// TwinCAT 3 PLC project LCLSVacuum
// Title: LCLSVacuumLib
// Company: SLAC
// Author: Alex Wallace & Scott Stubbs
// ProjectVersion: 1.12.0
// Description: No serial drivers exist in this library. Need LCLSVacuumSerialDrivers for that. 1.2.0 ecat diagnostic 1.2.1 added the ecat lib in here 1.2.2 adding the ratio check function for valve interlocking 1.3.6 added 275 & 500 gauges, minor changes 1.4.0 added a normally open gate valve structure and FB 1.5.0 added error and warning codes to ptm structure for pfeiffers 1.5.1 seamless override open/close on vgc during transition from override to normal mode. 1.7.0 ST_PTM now uses inheritence model. Started implementing Ebara support. 1.8.0 Moved to seperate functions for 937A and 937B controllers.
// ProgramVersion: 3.1.0.9
// libraries:
//   LCLS General,newest,SLAC
//   Tc2_EtherCAT, * (Beckhoff Automation GmbH)
//   Tc2_Standard, * (Beckhoff Automation GmbH)
//   Tc2_System, * (Beckhoff Automation GmbH)
//   Tc2_TcpIp, * (Beckhoff Automation GmbH)
//   Tc2_Utilities, * (Beckhoff Automation GmbH)
//   Tc3_Interfaces, * (Beckhoff Automation GmbH)
//   Tc3_Module, * (Beckhoff Automation GmbH)
// project tree:
//   Data types/Gauges/ E_PressureState.TcDUT, Gauge_Type.TcDUT, ST_VG.TcDUT
//   Data types/IO/ IO_EP2338.TcDUT
//   Data types/ ISG_Struct.TcDUT, ST_Encoder.TcDUT, UpStrInVac_Struct.TcDUT, UpStrOutVac_Struct.TcDUT
//   Data types/Pumps/ E_PumpState.TcDUT, ST_AgilentControlStatus.TcDUT, ST_AgilentPTM.TcDUT, ST_AuxiliaryPump.TcDUT, ST_EbaraDryPump.TcDUT, ST_EbaraPTM.TcDUT, ST_LeyboldPTM.TcDUT, ST_PfeifferPTM.TcDUT, ST_PIP.TcDUT, ST_PTM.TcDUT, ST_ReadbackOnlyPump.TcDUT, ST_RoughPump.TcDUT
//   Data types/Valves/ E_VCN.TcDUT, E_ValvePositionState.TcDUT, E_VGC.TcDUT, ST_VCC.TcDUT, ST_VCC_NO.TcDUT, ST_VCN.TcDUT, ST_VGC.TcDUT, ST_VGC_NO.TcDUT, ST_VRC.TcDUT
//   Global Variables/ Constants.TcGVL, Global_Variables.TcGVL
//   POUs/ Example_GaugeSup.TcPOU
//   POUs/Functions/Gauge FB/ FB_500.TcPOU, FB_903.TcPOU, FB_907.TcPOU, FB_275.TcPOU, FB_909.TcPOU, FB_925.TcPOU, FB_937A_VG.TcPOU, FB_937B_VG.TcPOU, FB_972.TcPOU, FB_Dumb_Gauge.TcPOU, FB_PressureState.TcPOU, FB_GCM.TcPOU, FB_GGO.TcPOU
//   POUs/Functions/Pumps/ FB_EbaraDryPump.TcPOU, FB_PTM_Pfeiffer.TcPOU, FB_PTM_Ebara.TcPOU, FB_PTM_Agilent.TcPOU, FB_PTM_MagDriveDigital.TcPOU, FB_PTM_LeyboldTD20Classic.TcPOU, FB_ScrollPump.TcPOU, FB_TurboExtLogic.TcPOU, FB_VARIAN301TURBO.TcPOU
//   POUs/Functions/Valve FB/ FB_TurbVentvalve_NO.TcPOU, FB_VCC_NO.TcPOU, FB_VCN.TcPOU, FB_VGC.TcPOU, FB_VGC_NO.TcPOU, FB_VRC.TcPOU, FB_VCC.TcPOU, FB_VRC_OK_CLS.TcPOU, F_VALVE_REL_ILK.TcPOU, F_VRC_DIODE_ILK.TcPOU, F_TURBO_VRC_ILK.TcPOU
//   Version/ Global_Version.TcGVL
// real-time tasks:
//   TASK PlcTask: cycle T#10ms, priority 20, ADS port 350
//   TASK LoggerTask: cycle T#10ms, priority 21, ADS port 351

// ---- Data types/Gauges/E_PressureState.TcDUT
TYPE E_PressureState :
(
	//Valid States (Positive)
	Valid := gc_GaugeValidState, // gc_GaugeValidState set in "Global Variable Folder: Constants"
	ValidHi	:= 1, 
	ValidLo	:= 2, 
	
	// Invalid states
	PressInvalid	:= -1, 
	GaugeDisconnected	:=	-2, 
	OoR	:= -6, 
	// Ion gauges
	Off		:= -3, 
	Starting	:= -4
) INT;
END_TYPE

// ---- Data types/Gauges/Gauge_Type.TcDUT
TYPE Gauge_Type: ( 
PG722B := 0, //Baraton Gauge
IG903 := 1 , //Cold Cathode
PG907 := 2 , //Pirani Gauge
IG909:= 3 , //Hot Cathode
PG925 := 4 ); //MicroPirani Gauge
(* This enumeration should match up with the EDM MUX button on the vacuum gauge expert controls screen *)
END_TYPE

// ---- Data types/Gauges/ST_VG.TcDUT
TYPE ST_VG :
STRUCT
	/// A general gauge structure is used to make the rest of the interlocking simpler. There are some parameters for cold cathodes that are not used by pirani.
	///These features aren't disabled, they just aren't used, think child/parent classes. 
	/// Readbacks 
	rPRESS: REAL; //This is the human-readable pressure
	iPRESS_R: INT; //input pressure in machine form
	xAT_VAC: BOOL; //Pressure At Vacuum
	xPRESS_OK: BOOL; // Pressure Reading is trustworthy
	eState	:	E_PressureState;
	
	/// Controls 
	xHV_DIS: BOOL;// Enable High Voltage when True
	xHV_SW: BOOL;// High Voltage Switch
	wHV_RO: WORD;// Relay Output Location
	 // Bakeout bit 
	xBAKEOUT: BOOL;
	//enum for gauge type - will replace iType
	eTYPE: Gauge_Type := Gauge_Type.PG907; 
	//Gauge type, deprecated (default to pirani)
	iTYPE: INT := 2;

	// Index location of the associated Pirani Gauge
	wPG: WORD;  
	
	xTurnOnTime: BOOL;/// Turn on Timers for cold cathode warmup 
	
	rVAC_SP: REAL := 0.5; // At vacuum setpoint for all gauges
	rPRO_SP: REAL := 0.01; // Protection setpoint for ion gauges at which the gauge turns off, not used for pirani
	rHYS_PR: REAL; // Protection setpoint hysteresis 
	rFULL_SCALE: REAL := 1000; // Full scale pressure in Torr for baratron pressure conversion 
END_STRUCT
END_TYPE

// ---- Data types/IO/IO_EP2338.TcDUT
TYPE IO_EP2338 :
STRUCT
	i_bInCh1	AT	%I*	:	BOOL;
	i_bInCh2	AT	%I*	:	BOOL;
	i_bInCh3	AT	%I*	:	BOOL;
	i_bInCh4	AT	%I*	:	BOOL;
	
	i_bInCh5	AT	%I*	:	BOOL;
	i_bInCh6	AT	%I*	:	BOOL;
	i_bInCh7	AT	%I*	:	BOOL;
	i_bInCh8	AT	%I*	:	BOOL;
	
	
	q_bInCh1	AT	%Q*	:	BOOL;
	q_bInCh2	AT	%Q*	:	BOOL;
	q_bInCh3	AT	%Q*	:	BOOL;
	q_bInCh4	AT	%Q*	:	BOOL;

	q_bInCh5	AT	%Q*	:	BOOL;
	q_bInCh6	AT	%Q*	:	BOOL;
	q_bInCh7	AT	%Q*	:	BOOL;
	q_bInCh8	AT	%Q*	:	BOOL;
END_STRUCT
END_TYPE

// ---- Data types/ISG_Struct.TcDUT
TYPE ISG_Struct :
STRUCT

	xdoHV1 : BOOL;
	xdoHV2 : BOOL;
	xdoHV3 : BOOL;

	xswHV1 : BOOL;
	xswHV2 : BOOL;
	xswHV3 : BOOL;

	xilkHV1 : BOOL;
	xilkHV2 : BOOL;
	xilkHV3 : BOOL;

END_STRUCT
END_TYPE

// ---- Data types/Pumps/E_PumpState.TcDUT
TYPE E_PumpState :
(
pumpSTOPPED	:= 0,
pumpSTARTING	:= 1,
pumpRUNNING	:= 2,
pumpFAULT := 3

);
END_TYPE

// ---- Data types/Pumps/ST_AgilentControlStatus.TcDUT
TYPE ST_AgilentControlStatus :
STRUCT

(* Inputs *)
	xdiR1   		:  BOOL;
	xdiLSpd 		:  BOOL;
	xdiStart		:  BOOL;
	xdiR2   		:  BOOL;
	xdiFlt   	:  BOOL;
	xswStart		:  BOOL;
	xswLSpd 		:  BOOL;
	xswSS   		:  BOOL;
	xilkStart	:  BOOL;
	xilkLSpd   	:  BOOL;
	xilkEnb   	:  BOOL;
	xilkSS   	:  BOOL;
	xAlmRst   	:  BOOL;

(* Outputs *)
	xdoStart	:  BOOL;
	xdoLSpd	:  BOOL;
	xdoEnb	:  BOOL;
	xdoSS	:  BOOL;

(* Alarm Outputs *)
	xalmFlt		:  BOOL;
	xalmStart	:  BOOL;
	xalmLSpd		:  BOOL;
	xalmSS		:  BOOL;
	xAlmSum		: BOOL;


END_STRUCT
END_TYPE

// ---- Data types/Pumps/ST_AgilentPTM.TcDUT
TYPE ST_AgilentPTM EXTENDS ST_PTM :
STRUCT

(* Inputs *)
	(* 24V in Ramp state; 0V for others *)
    i_xSTART :	BOOL; 
	
	(* setpoint related to frequency *)
	i_xR1	:  BOOL;
	
	(* setpoint related to Power *)
	i_xR2	:  BOOL;
	
	(* low speed mode *)
	i_xLSpd	:  BOOL;
	
	(* Fault input*)
	//i_xFault : BOOL;  Inherit ST_PTM.xFault
	
	

(* controls *)
	(* Start/Stop - 
		q_RunDo ;   Inherit ST_PTM.
	 *)
	
	(* Low speed control *)
	q_xLSpd		:  BOOL;
	
	(*Soft start *)
	q_xSS   	:  BOOL;
	
	(* Run interlock*)
	q_xIlk : BOOL;
		
	eState	:	E_PumpState;
	
	rForelinePressureSP : REAL := 0.01;
	rInletPressureSP : REAL := 0.5;
	

END_STRUCT
END_TYPE

// ---- Data types/Pumps/ST_AuxiliaryPump.TcDUT
TYPE ST_AuxiliaryPump EXTENDS ST_RoughPump :
STRUCT
	q_ContactClosed	:	BOOL;
END_STRUCT
END_TYPE

// ---- Data types/Pumps/ST_EbaraDryPump.TcDUT
TYPE ST_EbaraDryPump EXTENDS ST_RoughPump :
STRUCT
(* Extension of the rough pump archetype for ebara 
Applicable to: 
EV-S20
EV-S50
EV-S100
EV-S200
*)

//Controls
q_xMPStart	:	BOOL; //Main Pump start
q_xBPStart	:	BOOL; // Booster Pump start (this can be started by the pump automatically)

xBPIlk	:	BOOL;	//Booster pump interlock
rBPIlkSP	:	REAL := 30; //Booster pump pressure setpoint
tonBP	:	TON := (PT:=T#5S); //Timer for pressure and valve stability


//Readbacks
i_xMPStatus	:	BOOL; //MP status
i_xBPStatus	:	BOOL; //BP status
i_xWarning	:	BOOL; //Warning status
i_xAlarm	:	BOOL; //Alarm, maps to error
i_xRemote	:	BOOL; //Remote control status


END_STRUCT
END_TYPE

// ---- Data types/Pumps/ST_EbaraPTM.TcDUT
TYPE ST_EbaraPTM EXTENDS ST_PTM :
STRUCT
(* Extension of the PTM archetype for Ebara turbo controllers 
Applicable to: 
ETC series
*)
//Controls
i_xStart   : BOOL; //Momentary start switch
i_xStop    : BOOL; //Momentary stop switch
// i_xReset is momentary reset switch - resets protection functions

q_xStart   : BOOL; //Outputs - FB decides if these are actually set
q_xStop    : BOOL;
q_xReset   : BOOL;
q_xProtection : BOOL; //NC. If opened, pump will decelerate/not start

iq_xSpeedSet    : BOOL; //Request to set speed
q_iSpeedSet   : DINT; //Requested speed (min. 100 RPM)

i_xOverride   : BOOL; //Override mode - ignores interlocks

//Readbacks - also has Accel/At speed/Decel/Fault/Cur Speed (min 100RPM)
i_xRotate : BOOL; //If open, pump is rotating
i_xDecel  : BOOL; //If closed, brake engaged (pump decelerating)
i_xNCFault  : BOOL; //Normally closed fault wiring. If false, there is a fault, or cable is unplugged.
i_iRawSpeed	:	INT; //Raw pump speed from analog input

END_STRUCT
END_TYPE

// ---- Data types/Pumps/ST_LeyboldPTM.TcDUT
TYPE ST_LeyboldPTM EXTENDS ST_PTM :
STRUCT
(* Extension of the PTM archetype for Oerlikon turbo controllers 
Applicable to: 
Mag Drive Digital
Mag Drive S
More?
*)
//Readbacks
	i_xDecel	:	BOOL;
	i_diPumpTemp:	DINT;
	i_diPwr   	:   DINT;
	i_diElecTemp:	DINT;
	i_xTempFault:	BOOL;
	i_xNCError	:	BOOL; //Using normally closed wiring

//Controls
	q_xRemote : BOOL; (* Remote control enabled *)
END_STRUCT
END_TYPE

// ---- Data types/Pumps/ST_PfeifferPTM.TcDUT
TYPE ST_PfeifferPTM EXTENDS ST_PTM :
STRUCT
(* Extension of the PTM archetype for Pfeiffer turbos 
Applicable to: 
HiPace series w/ onboard controllers
More?
*)
//Readbacks
	i_diPwr		:	DINT;
	i_diElecTemp	:	DINT;
	i_diBtmTemp:	DINT;
	i_diBrngTemp:	DINT;
	i_diMtrTemp:	DINT;
	i_iErrorCode	:	INT; //might change these to enumeration someday
	i_iWarningCode	:	INT;
	i_xTempFault	:	BOOL;
	i_uiPowerPctRbk :   UINT;
	
//Controls
	q_uiPowerPct : UINT := 100; //Should normally be 100
	
END_STRUCT
END_TYPE

// ---- Data types/Pumps/ST_PIP.TcDUT
TYPE ST_PIP :
STRUCT
(* Interlock *)
   xHV_ExtIlk : BOOL; 

	rHVEna_SP : REAL := 1.0E-4;	
	
(* EPICS Controls *)	
	i_xHVEna_SW : BOOL; 
	
(* Controls *)
	q_xHVEna_DO : BOOL;	



END_STRUCT
END_TYPE

// ---- Data types/Pumps/ST_PTM.TcDUT
TYPE ST_PTM :
STRUCT
(* General PTM Structure
Each PTM might have a serial control structure, but all will have a general supervisory control structure

NOTE: This is an archetype, use an extension of this structure for a specific pump (or make one).

*)

(* Controls *)
	i_xRunSW	:	BOOL;
	i_xReset	:	BOOL; //For resetting faults
	q_RunDO 	:	BOOL;

(* Readbacks *)
	xExtRunOk	:	BOOL; (* also a control *)
	i_xAccel	:	BOOL;
	i_xAtSpd	:	BOOL;
	i_diCurSpd	:	DINT;
	
	xCommTimeout	:	BOOL := TRUE;  (* Initialized true since we haven't talked to pump yet *)
(* Alarm Outputs *)
	xFault		:	BOOL; //Note, for Ebara this is *false* in a fault condition!
	xWarn		:	BOOL; (* warning *)
	
(* IWS instructions *)
	xActive	:	BOOL; // this bit is set to add the pump to the system
	iPumpGrp 	:	INT; // all members of a pump group start at the same time
	
(* Operational Setpoints *)
	rForelineSP	:	REAL := 0.5;

END_STRUCT
END_TYPE

// ---- Data types/Pumps/ST_ReadbackOnlyPump.TcDUT
//Simple type for a pump where we have readback only, no control.

TYPE ST_ReadbackOnlyPump :
STRUCT
	i_xPumpOn : BOOL;
	i_diPumpSpeed : DINT; //Arbitrary
END_STRUCT
END_TYPE

// ---- Data types/Pumps/ST_RoughPump.TcDUT
TYPE ST_RoughPump :
STRUCT
	
(* Generic roughing pump controls 

NOTE: This is an archetype, use an extension of this structure for a specific pump (or make one).

*)

//Controls
i_xRunSW	:	BOOL; //epics/ software control switch
q_xRunDo 	:   BOOL; 

//Status and Readback
xIlk	:	BOOL; //Interlock bit, true means OK to run
xExtIlk	:	BOOL; //External interlock, this is where the logic goes
xAtSpd	:	BOOL; //Pump at speed setpoint

xWrn	:	BOOL; //Pump warning
iWrn	:	BOOL; //Warning state/code
xErr	:	BOOL; //Error summary
iErr	:	BOOL; //Error state/code

END_STRUCT
END_TYPE

// ---- Data types/ST_Encoder.TcDUT
TYPE ST_Encoder :
STRUCT
	xENC_PWR_SW : BOOL;
	xENC_PWR : BOOL;
END_STRUCT
END_TYPE

// ---- Data types/UpStrInVac_Struct.TcDUT
TYPE UpStrInVac_Struct :
STRUCT

	xdiUpSVac : BOOL;

END_STRUCT
END_TYPE

// ---- Data types/UpStrOutVac_Struct.TcDUT
TYPE UpStrOutVac_Struct :
STRUCT

	xdoUpSVac : BOOL;
	xilkUpSVac : BOOL;

END_STRUCT
END_TYPE

// ---- Data types/Valves/E_VCN.TcDUT
TYPE E_VCN :
	(
		CloseValve		:= 0,
		OpenValve		:= 2
	);
END_TYPE

// ---- Data types/Valves/E_ValvePositionState.TcDUT
TYPE E_ValvePositionState :
	(
OPEN	:= 0,
CLOSED	:= 1,
MOVING	:= 2,
INVALID :=3
	);
END_TYPE

// ---- Data types/Valves/E_VGC.TcDUT
TYPE E_VGC :
(

	Vented,
	AtVacuum,
	ERR_DiffPress,
	ERR_LostVac

);
END_TYPE

// ---- Data types/Valves/ST_VCC.TcDUT
TYPE ST_VCC :
STRUCT

(* Inputs *)
	xOPN_SW	: BOOL;
	xOvrdOpn	:	BOOL;
	xOPN_OK	: BOOL;

(* Outputs *)
	xOPN_DO	: BOOL;

END_STRUCT
END_TYPE

// ---- Data types/Valves/ST_VCC_NO.TcDUT
TYPE ST_VCC_NO :
STRUCT

(* A normally open valve needs permission to close! *)
(* Inputs *)
	xCLS_SW	: BOOL;
	xOvrdCls	:	BOOL;
	xCLS_OK	: BOOL;

(* Outputs *)
	xCLS_DO	: BOOL;

END_STRUCT
END_TYPE

// ---- Data types/Valves/ST_VCN.TcDUT
TYPE ST_VCN :
STRUCT
	(* VCN - Valve Controlled Needle
	Used for Pfeiffer EVR 116 needle valves *)
	// Inputs
	i_iPosition	:	INT; //Position readback (if it exists)
	
	// Outputs
	q_iRawPosition	:	INT; //Position control 
	//For the EVR 116 this is 0-10V analog
	
	//Softvariables
	xIlk	:	BOOL := FALSE; // Interlock Bit
	rUpperLimit	:	REAL;	//Upper limit on valve open
	rReqPosition	:	REAL; //Requested position (0.0-100.0%)
	eValveControl	:	E_VCN := E_VCN.CloseValve; // Valve control state

	ftIlk	:	F_TRIG;	

END_STRUCT
END_TYPE

// ---- Data types/Valves/ST_VGC.TcDUT
TYPE ST_VGC :
STRUCT

(* Readbacks *)
	i_xOpnLS	: BOOL;
	i_xClsLS	: BOOL;

(* EPICS Controls *)
	xOPN_SW	: BOOL;
	xAlmRst	: BOOL;
	xOvrdOpn	:	BOOL;

(* Interlocks *)
	xDP_OK	:	BOOL;	// Indicates the valve can be opened because the differential pressure is low enough
	xEXT_OK	:	BOOL := FALSE;	(* External interlock for custom interlocking in addition to regular DP ilk, this must be set true, or the interlock condition before calling the FB_VGC *)
	xOPN_OK	:	BOOL;	(* Final SUM of DP_OK and EXT_OK, needed because it allows the DP ilk to be switched off, see FB_VGC.Dis_DPIlk *)
	
	rAT_VAC_SP	:	REAL := 0.01;	// Interlock setpoint for gauges on both sides of valve
	rAT_VAC_SP_LAST	:	REAL :=0.01 ;	// Interlock setpoint for gauges on both sides of valve
	rAT_VAC_HYS	:	REAL :=0.01;	// Hysteresis of the vacuum sp
	rHYST_PERC	:	REAL := 0.80;	// Hysteresis percentage
	xAT_VAC	:	BOOL;	//At vacuum setpoint
	
eState	:	E_ValvePositionState := E_ValvePositionState.INVALID;
(* Controls *)
	xOPN_DO	: BOOL;

(* Alarm Outpus *)
	xERR_DifPres		: 	BOOL;
	xERR_LstVac		: 	BOOL;
	xERR_SM		:	BOOL; //Issue with the valve state-machine. This state should be excluded, if this boolean is true, something dramatic in the PLC software has happened.
	xAlmSum			: 	BOOL;

END_STRUCT
END_TYPE

// ---- Data types/Valves/ST_VGC_NO.TcDUT
TYPE ST_VGC_NO EXTENDS ST_VGC :
STRUCT
	(* A normally open gate valve needs permission to close! *)
	(* EPICS Controls *)
	xCLS_SW	:	BOOL;
	xOvrdCls	:	BOOL;
	
	(* Interlocks *)
	xCLS_OK	:	BOOL;
	
	(* IO Controls *)
	xCLS_DO	:	BOOL;
	
	
END_STRUCT
END_TYPE

// ---- Data types/Valves/ST_VRC.TcDUT
TYPE ST_VRC :
STRUCT
(* Readbacks *)
	//If True, Valve is Open
	i_xOpnLS	:	BOOL;
	//If True, Valve is Closed
	i_xClsLS	:	BOOL;
	
	eState	:	E_ValvePositionState := E_ValvePositionState.INVALID;

(* Inputs *)
	//Manually Pressing valve "Open/Close" on EDM
	xOPN_SW	: BOOL;
	//Manually toggling valve Local "ILK on button" on EDM
	xOvrdOpn	:	BOOL;
	//Calculated permissions to open valve
	xOPN_OK	: BOOL;
	//In case VRC is normally open
	xCLS_OK : BOOL := TRUE;
(* Outputs *)
	//When True, Opens valve
	//When False, Closes valve
	xOPN_DO	: BOOL;

END_STRUCT
END_TYPE

// ---- Global Variables/Constants.TcGVL
VAR_GLOBAL CONSTANT
	gc_iSizeOfGGOArray : INT := 50;
	gc_GaugeValidState :	INT := 0;
END_VAR

// ---- Global Variables/Global_Variables.TcGVL
VAR_GLOBAL
	g_stSystem	:	System_Struct:= (
    	xFirstScan := TRUE
	);
	
	g_DummyVG	:	ST_VG;
	
END_VAR

// ---- Version/Global_Version.TcGVL
{attribute 'TcGenerated'}
// This function has been automatically generated from the project information.
VAR_GLOBAL CONSTANT
	{attribute 'const_non_replaced'}
	{attribute 'linkalways'
	stLibVersion_LCLSVacuumLib : ST_LibVersion := (iMajor := 1, iMinor := 12, iBuild := 0, iRevision := 0, sVersion := '1.12.0');
END_VAR

// ---- POUs/Example_GaugeSup.TcPOU
PROGRAM Example_GaugeSup
VAR

	LMP_VG00	:	ST_VG; (* simulation pirani *)

	fb_LMP_VG :	FB_GGO;
	i : INT;

END_VAR

(* Dummy pirani setup *)
LMP_VG00.rPRESS_OK := TRUE;

(* The following condition ensures that the pressure switches to the GPI:20 when VRC 06 is closed and VRC 05 is open *)

(* Changed interlock here to GPI 20 for running without the GPI 30 gauge *)
(*
IF LMP_VRC05.OPN-DO AND NOT LMP_VRC06.OPN_DO THEN
fb_LMP_GPI_D1(PG := LMP_GPI_D1, PGA := LMP_GPI20, PGB := LMP_GPI01, VICA := LMP_VRC05, VICB := LMP_VRC02);
ELSE
fb_LMP_GPI_D1(PG := LMP_GPI_D1, PGA := LMP_GPI30, PGB := LMP+GPI01, VICA := LMP_VRC06, VICB := LMP_VRC02);
END_IF
*)
(* Dumb Gauge *)
(* fb_LMP_GPI_D1 (PG := LMP_GPI_D1, PGA := LMP_GPI20, PGB := LMP_GPI01, VICA := LMP_VRC05, VICB := LMP_VRC02); *)

LMP_VG[20].VAC_SP := 7.5;
LMP_VG[1].VAC_SP := 1E-1;
LMP_VG[2].VAC_SP := 1E-1;
LMP_VG[12].VAC_SP := 5E-7;

(* Upstream vacuum OK signal *)
(* This signal tells the AMO_PLC that the KBP_VGC_02 is OK to open *)
DiscIO_IC_EB1Ch08 := LMP_VG[12].AT_VAC AND LMP_VGC10.OPN_LS;

(* pnCCD Chamber *)
LMP_VG[40].FULL_SCALE := 1000;
LMP_VG[41].FULL_SCALE := 1;

LMP_VG[1].GAUGE := PG925;
LMP_VG[2].GAUGE := PG925;
LMP_VG[10].GAUGE := PG907;
LMP_VG[11].GAUGE := PG907;
LMP_VG[12].GAUGE := IG903;
LMP_VG[13].GAUGE := IG909;
LMP_VG[20].GAUGE := PG907;
LMP_VG[21].GAUGE := IG903;
LMP_VG[22].GAUGE := IG909;
LMP_VG[30].GAUGE := PG907;
LMP_VG[31].GAUGE := IG903;
LMP_VG[40].GAUGE := PG722B;
LMP_VG[41].GAUGE := IG903;
LMP_VG[42].GAUGE := PG722B;
LMP_VG[43].GAUGE := IG909;

FOR i := 1 TO 50 DO
fb_LMP_VG (index := i, astGauges := LMP_VG);
END_FOR

(*
(* Control function blocks *)

(* Roughing lines *)
fb_LMP_VG01(PG := LMP_VG[1]); (* roughing line *)
fb_LMP_VG02(PG := LMP_VG[2]); (* roots line *)

(* Differential Pumping Chambers *)
(* fb_LMP_GCC10 (IG := LMP_GCC10, PG := LMP_GPI00); *)
(* fb_LMP_GCC11 (IG := LMP_GCC11, PG := LMP_GPI00); *)
fb_LMP_VG10 (PG := LMP_VG[10]);
fb_LMP_VG11 (PG := LMP_VG[11]);

(* Interaction Chamber *)
fb_LMP_VG21 (IG := LMP_VG[21], PG := LMP_VG[20]);
fb_LMP_VG22 (IG := LMP_VG[22], PG := LMP_VG[20]);
fb_LMP_VG20 (PG := LMP_VG[20]);

(* Upstream vacuum OK signal *)
(* This signal tells the AMO_PLC that the KBO_VGC_02 is OK to open *)
DiscIO_IC_EB1Ch08 := LMP_VG[12].AT_VAC AND LMP_VGC10.OPN_LS;

(* Detector Chamber *)
fb_LMP_VG31 (IG := LMP_VG[31], PG := LMP_VG[30]);
fb_LMP_VG30 (PG := LMP_VG[30]);

(* pnCCD Chamber *)
fb_LMP_VG41 (IG := LMP_VG[41], PG := LMP_VG[40]);
fb_LMP_VG43 (IG := LMP_VG[43], PG := LMP_VG[42]);
LMP_VG[40].FULL_SCALE := 1000;
LMP_VG[41].FULL_SCALE := 1;
fb_LMP_VG40 (PG := LMP_VG[40]);
fb_LMP_VG42 (PG := LMP_VG[42]);
*)

END_PROGRAM

// ---- POUs/Functions/Gauge FB/FB_GGO.TcPOU
FUNCTION_BLOCK FB_GGO
VAR_IN_OUT
	iq_astGauges: ARRAY[0..gc_iSizeOfGGOArray] OF ST_VG;
	iq_axHV_RO: ARRAY[0..gc_iSizeOfGGOArray] OF BOOL;
END_VAR
VAR_INPUT
	i_iIndex: INT;
END_VAR
VAR

	stPG: ST_VG;
	stVG: ST_VG;
	//index for associated pirani
	wPG : WORD;

	
	// FBs
	fb903	:	FB_903;
	fb907	:	FB_907;
	fb909	:	FB_909;
	fb925	:	FB_925;
	fbGCM	:	FB_GCM;
	
END_VAR

(* This function block is used to calculate the pressure from the analog input voltage and to provide protection and automatic turn on of ion gauges.
 It also manages the turn on fo the AT_VAC boolean, and checks to make sure the pressure is good *)

(* Full-scale pressure conversion factor *)

(* Real-value voltage calculation *)
(* Generic expression for pressure in the MKS systems

P = 10^(V/0.6-12)

722B = 0
903 = 1
907 = 2
909 = 3
925 = 4

*)

(* Make a copy of gauge at index*)
stVG := iq_astGauges[LIMIT(0 ,i_iIndex, gc_iSizeOfGGOArray)];

(* Check that it is an ion gauge *)
IF stVG.eTYPE = Gauge_Type.IG903 OR stVG.eTYPE = Gauge_Type.IG909 THEN

(* Check that Associated Gauge is within index*)
	IF WORD_TO_INT(stVG.wPG) <= gc_iSizeOfGGOArray THEN
		(* Check pressure gauge type before assignment *)
		(* Add high pressure gauge types here *)
		IF iq_astGauges[stVG.wPG].eTYPE = PG722B OR //722B
		iq_astGauges[stVG.wPG].eTYPE = PG907 OR //907
		iq_astGauges[stVG.wPG].eTYPE = PG925 THEN //925
			stPG := iq_astGauges[stVG.wPG];  (* Copy associated pirani gauge number to local variable *)
		ELSE //Default to allow the IG to turn on, this allows someone to set the PG to another IG and turn the gauge on whenever they want
			stPG.rPRESS := 1E-3;
			stPG.xPRESS_OK := TRUE;
		END_IF
	
	END_IF
END_IF

(* Evaluate each Gauge pressure based on eTYPE*)
CASE iq_astGauges[i_iIndex].eTYPE OF
	
	//Baratron Gauge
	PG722B:
		fbGCM(VG:=iq_astGauges[i_iIndex]);
		
	//Cold Cathode
	Gauge_Type.IG903:
		fb903(IG:=iq_astGauges[i_iIndex], PG:=iq_astGauges[wPG]);
		
	//Pirani Gauge	
	PG907:
		fb907(PG:=iq_astGauges[i_iIndex]);
		
	//Hot Cathode	
	Gauge_Type.IG909:
		fb909(IG:=iq_astGauges[i_iIndex], PG:=iq_astGauges[wPG]);
		
	//MicroPirani Gauge	
	PG925:
		fb925(PG:=iq_astGauges[i_iIndex]);
	ELSE
		(* Now, since we don't know what gauge type we're dealing with, we want 
		to make sure to reset all the gauge parameters, otherwise we may be 
		left with stale information *)
	stVG.rPRESS := 760;
	stVG.xAT_VAC := FALSE;
	stVG.xPRESS_OK := FALSE;
	stVG.xHV_SW := FALSE;
		
END_CASE

(* reAssign "HV On" back into High Voltage Array*)
iq_axHV_RO[LIMIT(0,WORD_TO_INT(stVG.wHV_RO),gc_iSizeOfGGOArray)]:=stVG.xHV_DIS;

END_FUNCTION_BLOCK

// ---- POUs/Functions/Gauge FB/FB_903.TcPOU
FUNCTION_BLOCK FB_903
VAR_IN_OUT

	IG : ST_VG;

END_VAR
VAR_INPUT

	PG : ST_VG;

END_VAR
VAR_OUTPUT
END_VAR
VAR
	rMaxPressure: REAL := 5E-3;
	rMinPressure: REAL := 5E-11; (* Even though spec is 3E-10, manual states that the discharge is off only if output voltage is <0.5V. 
                                    Since this corresponds to ~3.2E-11 torr, let's be safe and call the min. 5E-11. *)

	V: LREAL;
	fbGaugeState : FB_PressureState;
END_VAR

(* This function block is used to provide protection and automatic turn on of ion gauges,
 it also manages the turn on of the AT_VAC boolean, and checks to make sure the pressure is good *)

(* Real-value calculation *)
(* Generic expression for pressure in the MKS systems

P = 10^(V/0.6 -12)

*)

V := 10*INT_TO_LREAL(IG.iPRESS_R)/32767;

IG.rPRESS := LREAL_TO_REAL(EXPT(10,(V-11)));


(* Protection Functions *)
(* If the PG pressure is greater than the IG.PRO_SP then the gauge is disabled *)
(* If the PG pressure is less than the IG.PRO_SP then the gauge is enabled *)
(* This FB also implements some hysteresis so the gauge doesn't have rapid power cycling while near the turn on boundary *)

IF PG.rPRESS <= IG.rPRO_SP AND PG.xPRESS_OK THEN

	IG.xHV_DIS := IG.xHV_SW;

ELSIF IG.xHV_DIS THEN
	IF (IG.rPRESS > (IG.rPRO_SP + IG.rHYS_PR)) OR PG.rPRESS > (IG.rPRO_SP + IG.rHYS_PR) THEN
		IG.xHV_DIS := FALSE;
		IG.xHV_SW := FALSE;
	END_IF
ELSE
	IG.xHV_DIS := FALSE;
	IG.xHV_SW := FALSE;
END_IF

(* Pressure OK check *)
fbGaugeState.i_rV := V;
fbGaugeState.i_MaxPressure := rMaxPressure;
fbGaugeState.i_MinPressure := rMinPressure;
fbGaugeState(iq_stVG:=IG);

//Backwards compatibility
IG.xPRESS_OK := (IG.eState = Valid) OR IG.xBAKEOUT;

(* Setpoint evaluation *)
IG.xAT_VAC := (IG.xPRESS_OK AND (IG.rPRESS<IG.rVAC_SP)) OR IG.xBAKEOUT;

END_FUNCTION_BLOCK

// ---- POUs/Functions/Gauge FB/FB_PressureState.TcPOU
FUNCTION_BLOCK FB_PressureState
VAR_INPUT
	i_rV	:	REAL;
	i_rVMin	:	REAL := 0.01; // Anything less than this voltage is considered disconnected
	i_rVMax :	REAL := 10.5; // Anything more than this is considered invalid
	i_IGTurnOnTime	:	TIME := T#10S;
	
	i_MinPressure	:	REAL;
	i_MaxPressure	:	REAL;
END_VAR
VAR_OUTPUT
	q_eState 	:	E_PressureState;
END_VAR
VAR_IN_OUT
	iq_stVG	:	ST_VG;
END_VAR
VAR
	tonGaugeTurnOnTmr : TON;
END_VAR

(* Pressure State Evaluation
A. Wallace, 2016-8-31

This FB serves to evaluate the state of the pressure based on the raw voltage, pressure, and gauge state.

*)
// Is the gauge plugged in, and within a reasonable range?
IF i_rV < i_rVMin THEN
	q_eState := E_PressureState.GaugeDisconnected;
ELSIF i_rV > i_rVMax THEN
	q_eState := E_PressureState.PressInvalid;
ELSE
	// Is the gauge reading back a pressure that makes sense?
	CASE iq_stVG.eTYPE OF
		Gauge_Type.IG903:
			tonGaugeTurnOnTmr(IN:=iq_stVG.xHV_DIS, PT:=i_IGTurnOnTime, Q=>iq_stVG.xTurnOnTime);
			IF iq_stVG.xHV_DIS THEN
				IF tonGaugeTurnOnTmr.Q THEN
					IF iq_stVG.rPRESS >= i_MinPressure AND iq_stVG.rPRESS <= i_MaxPressure THEN
						q_eState := E_PressureState.Valid;
					ELSE
						q_eState := OoR; 
					END_IF
				ELSE
						q_eState := E_PressureState.Starting;
				END_IF
			ELSE
				q_eState := E_PressureState.Off;
			END_IF
		Gauge_Type.IG909:
			IF iq_stVG.xHV_DIS THEN
				IF iq_stVG.rPRESS >= i_MinPressure AND iq_stVG.rPRESS <= i_MaxPressure THEN
					q_eState := E_PressureState.Valid;
				ELSE
					q_eState := E_PressureState.OoR;
				END_IF
			ELSE
				q_eState := E_PressureState.Off;
			END_IF
		Gauge_Type.PG907, Gauge_Type.PG925, Gauge_Type.PG722B:
			IF iq_stVG.rPRESS >= i_MinPressure AND iq_stVG.rPRESS <= i_MaxPressure THEN
				q_eState := E_PressureState.Valid;
			ELSIF iq_stVG.rPRESS < i_MinPressure THEN
				q_eState := E_PressureState.ValidLo;
			ELSE
				q_eState := E_PressureState.ValidHi;
			END_IF
		ELSE
			q_eState := E_PressureState.PressInvalid;
	END_CASE
END_IF


iq_stVG.eState := q_eState;

// Legacy Press OK boolean eval
iq_stVG.xPRESS_OK := q_eState >= gc_GaugeValidState;

END_FUNCTION_BLOCK

// ---- POUs/Functions/Gauge FB/FB_907.TcPOU
FUNCTION_BLOCK FB_907
VAR_IN_OUT

	PG : ST_VG;

END_VAR
VAR_INPUT
END_VAR
VAR_OUTPUT
END_VAR
VAR
	V : LREAL;
	fbGaugeState : FB_PressureState;
END_VAR
VAR CONSTANT
	A : LREAL := 3.29;
	B : LREAL := 24.98;
	C : LREAL  := 0.98;
	V_0 : LREAL := 0.3752;
	D: LREAL := 4.929;
	F: LREAL := 1.6E-6;
	G: LREAL := -225;
	H: LREAL := 2.0253;
	K: LREAL := 0.52703;
	
	// Torr
	rMaxPressure: REAL := 1000;
	// Torr
	rMinPressure: REAL := 1E-3;
END_VAR

(* This function block is used to provide protection and automatic turn on of ion gauges,
 it also manages the turn on of the AT_VAC boolean, and checks to make sure the pressure is good *)

 //Default setpoint 50 mT
IF PG.rVAC_SP = 0 THEN
	PG.rVAC_SP := 5E-2;
END_IF
 
(* Real-value calculation *)

V := 10*INT_TO_LREAL(PG.iPRESS_R)/32767;

IF V > 0.38 AND V < 4.85 THEN

PG.rPRESS := LREAL_TO_REAL(EXPT((A/(B/(EXPT(V,2)-EXPT(V_0,2)-1))), 1/C));

ELSIF V > 4.85 AND V < 5.18 THEN

PG.rPRESS := LREAL_TO_REAL(SQRT( ( (V-D)+SQRT(EXPT((V-D),2)-4*F*G ))/(2*F) ));

ELSIF V> 5.18 THEN

PG.rPRESS := LREAL_TO_REAL(EXP((V-H)/K));

END_IF

(* Pressure OK check *)
fbGaugeState.i_rV := LREAL_TO_REAL(V);
fbGaugeState.i_MaxPressure := rMaxPressure;
fbGaugeState.i_MinPressure := rMinPressure;
fbGaugeState(iq_stVG:=PG);


(* Setpoint evaluation *)
PG.xAT_VAC := PG.xPRESS_OK AND (PG.rPRESS<PG.rVAC_SP) OR PG.xBAKEOUT;

END_FUNCTION_BLOCK

// ---- POUs/Functions/Gauge FB/FB_909.TcPOU
FUNCTION_BLOCK FB_909
VAR_IN_OUT

	IG : ST_VG;

END_VAR
VAR_INPUT

	PG : ST_VG;

END_VAR
VAR_OUTPUT
END_VAR
VAR
	rMaxPressure: REAL := 5E-2;
	rMinPressure: REAL := 3E-10;

	V: REAL;
	fbGaugeState : FB_PressureState;
END_VAR

(* This function block is used to provide protection and automatic turn on of ion gauges,
 it also manages the turn on of the AT_VAC boolean, and checks to make sure the pressure is good *)

(* Real-value calculation *)
(* Generic expression for pressure in the MKS systems

P = 10^(V/0.6 -12)

*)

V := 10*INT_TO_REAL(IG.iPRESS_R)/32767;

IG.rPRESS := LREAL_TO_REAL(EXPT(10,(V-10)));


(* Protection Functions *)
(* If the PG pressure is greater than the IG.PRO_SP then the gauge is disabled *)
(* If the PG pressure is less than the IG.PRO_SP then the gauge is enabled *)
(* This FB also implements some hysteresis so the gauge doesn't have rapid power cycling while near the turn on boundary *)

IF PG.rPRESS <= IG.rPRO_SP AND PG.xPRESS_OK THEN

	IG.xHV_DIS := IG.xHV_SW;

ELSIF IG.xHV_DIS THEN
	IF IG.rPRESS > IG.rPRO_SP + IG.rHYS_PR OR PG.rPRESS > IG.rPRO_SP + IG.rHYS_PR THEN
		IG.xHV_DIS := FALSE;
		IG.xHV_SW := FALSE;
	END_IF
ELSE
	IG.xHV_DIS := FALSE;
	IG.xHV_SW := FALSE;
END_IF

(* Pressure OK check *)
fbGaugeState.i_rV := V;
fbGaugeState.i_MaxPressure := rMaxPressure;
fbGaugeState.i_MinPressure := rMinPressure;
fbGaugeState(iq_stVG:=IG);

//Backwards compatibility
IG.xPRESS_OK := (IG.eState = Valid) OR IG.xBAKEOUT;

(* Setpoint evaluation *)
IG.xAT_VAC := (IG.xPRESS_OK AND (IG.rPRESS<IG.rVAC_SP)) OR IG.xBAKEOUT;

END_FUNCTION_BLOCK

// ---- POUs/Functions/Gauge FB/FB_925.TcPOU
FUNCTION_BLOCK FB_925
VAR_INPUT
END_VAR
VAR_OUTPUT
END_VAR
VAR_IN_OUT
	PG	: ST_VG;
END_VAR
VAR
	rV : REAL;
	fbGaugeState : FB_PressureState;
	rMaxPressure	:	REAL := 760; //Torr
	rMinPressure	:	REAL := 1E-5; //Torr
END_VAR

(* Standard MKS 9XX series conversion *)
(* works for 972 and 925 *)

//Default setpoint 50 mT
IF PG.rVAC_SP = 0 THEN
	PG.rVAC_SP := 5E-2;
END_IF

rV := 10*INT_TO_REAL(PG.iPRESS_R)/32767;

IF rV >= 0.99 THEN
	IF rV >= 0.99 AND rV < 1 THEN
		PG.rPRESS := 1E-5;
	ELSE
		PG.rPRESS := LREAL_TO_REAL(EXPT(10, REAL_TO_LREAL(rV-6)));
	END_IF
	PG.xPRESS_OK := TRUE; //Backwards compatibility
ELSE
	PG.xPRESS_OK := FALSE;
END_IF

(* Pressure OK check *)
fbGaugeState.i_rV := rV;
fbGaugeState.i_MaxPressure := rMaxPressure;
fbGaugeState.i_MinPressure := rMinPressure;
fbGaugeState(iq_stVG:=PG);

(* Setpoint evaluation *)
PG.xAT_VAC := PG.xPRESS_OK AND (PG.rPRESS < PG.rVAC_SP);

END_FUNCTION_BLOCK

// ---- POUs/Functions/Gauge FB/FB_GCM.TcPOU
FUNCTION_BLOCK FB_GCM
VAR_IN_OUT
	VG	:	ST_VG;
END_VAR
VAR_OUTPUT
END_VAR
VAR
	rMinPressure: REAL;
	rV	:REAL;
END_VAR

(* Baratron Pressure Calc 
A. Wallace
2016-6-16
The full-scale pressure times the ratio of the meas.
voltage to full-scale voltage (10V).
The minimum pressure is always going to be 5e-4 * F.S.V.*)

rMinPressure := VG.rFULL_SCALE * 5E-4;


rV :=MAX((10*INT_TO_REAL(VG.iPRESS_R)/32767),0);
VG.rPRESS := (VG.rFULL_SCALE/10)*rV;
IF VG.rPRESS > rMinPressure THEN
	VG.xPRESS_OK := TRUE;
ELSE
	VG.xPRESS_OK := FALSE;
END_IF

END_FUNCTION_BLOCK

// ---- POUs/Functions/Gauge FB/FB_500.TcPOU
FUNCTION_BLOCK FB_500
VAR_IN_OUT
	IG : ST_VG;
END_VAR
VAR_INPUT
	PG	:	ST_VG;
END_VAR
VAR_OUTPUT
	xHV_SW: BOOL;
	rPRESS: INT;
	rVAC_SP: INT;
END_VAR
VAR
	rV : REAL;
	GaugeTurnOnTmr : TON;
	MinPressure: REAL := 1E-10;
	
END_VAR
VAR CONSTANT
	cDefaultPressure : REAL := 750.0;
	vBase	:	REAL := 0; //corresponding vbase 0V based on default curve.  See manual pg. 44
	pBase	:	REAL := 1.0E-10; //default curve base pressure is 1E-10. Confusing since can't actually read that low using analog out.
	vSlope	:	REAL := 1.0; //looks correct for default curve
END_VAR

(* 500 Logarithmic Output Conversion, factory default configuration *)

rV := 10*INT_TO_REAL(IG.iPRESS_R)/32767;

IF rV >= 0.49 AND rV < 0.6  THEN
	IG.eState := E_PressureState.Starting;
	IG.rPRESS := cDefaultPressure;
ELSIF rV < 0.4 THEN
	IG.eState := E_PressureState.Off;
	IG.rPRESS := cDefaultPressure;
ELSE
	IG.eState := E_PressureState.Valid;
	IG.rPRESS := LREAL_TO_REAL(EXPT(10,((rV-vBase)/vSlope+LOG(pBase))));
END_IF



(* Ion Gauge Protection Functions *)
(* If the PG pressure is greater than the VG.PRO_SP then the gauge is disabled *)
(* If the PG pressure is less than the VG.PRO_SP then the gauge is enabled *)
(* This FB also implements some hysteresis so the gauge doesn't have rapid power cycling while near the turn on boundary *)

IF PG.rPRESS <= IG.rPRO_SP AND PG.xPRESS_OK THEN

	IG.xHV_DIS := IG.xHV_SW;

ELSIF IG.xHV_DIS THEN
	IF IG.rPRESS > (IG.rPRO_SP + IG.rHYS_PR)  OR PG.rPRESS > (IG.rPRO_SP + IG.rHYS_PR) THEN
		IG.xHV_DIS := FALSE;
		IG.xHV_SW := FALSE;
	END_IF
ELSE
	IG.xHV_DIS := FALSE;
	IG.xHV_SW := FALSE;
END_IF

(* Pressure gauge OK checks *)

//Backwards compatibility
IG.xPRESS_OK := (IG.eState = E_PressureState.Valid) OR IG.xBAKEOUT;

(* Setpoint evaluation *)
IG.xAT_VAC := (IG.xPRESS_OK AND (IG.rPRESS < IG.rVAC_SP)) OR IG.xBAKEOUT;

END_FUNCTION_BLOCK

// ---- POUs/Functions/Gauge FB/FB_275.TcPOU
FUNCTION_BLOCK FB_275
VAR_IN_OUT
	PG : ST_VG;
END_VAR
VAR_INPUT
END_VAR
VAR_OUTPUT
END_VAR
VAR

	MinPressure: REAL := 1E-4;

	V : REAL;

	Vlowest: REAL := 10;
END_VAR
VAR CONSTANT
	rValidLoBoundary	:	REAL := 0.38;
	rDisconnectedBoundary	:	REAL := 0.3;
END_VAR

(* This function block is used to provide protection and automatic turn on of ion gauges,
 it also manages the turn on of the AT_VAC boolean, and checks to make sure the pressure is good *)
(* For MKS 275 mini-convectron *)

 //Default setpoint 50 mT
IF PG.rVAC_SP = 0 THEN
	PG.rVAC_SP := 5E-2;
END_IF

(* Real-value calculation *)

V := 10*INT_TO_REAL(PG.iPRESS_R)/32767;	

Vlowest := MIN(V, Vlowest);

IF V > rDisconnectedBoundary AND V <= rValidLoBoundary THEN

PG.rPRESS := MinPressure;
PG.eState := ValidLo;

ELSIF V > rValidLoBoundary AND V < 2.842 THEN

PG.rPRESS := MAX( MinPressure, LREAL_TO_REAL( -0.02585 + 0.03767*V + 0.04563*EXPT(V,2)+ 0.1151*EXPT(V,3) - 0.04158*EXPT(V,4)+ 0.008737*EXPT(V,5)) );
PG.eState := Valid;

ELSIF V >= 2.842 AND V < 4.945 THEN

PG.rPRESS := LREAL_TO_REAL((0.1031-0.02322*V+0.07229*EXPT(V,2))/(1-0.3986*V+0.07438*EXPT(V,2)-0.006866*EXPT(V,3)));
PG.eState := Valid;

ELSIF V >= 4.945 AND V < 5.659 THEN

PG.rPRESS := LREAL_TO_REAL((100.624-20.5623*V)/(1-0.37679*V+0.0348656*EXPT(V,2)));
PG.eState := Valid;

ELSIF V <= rDisconnectedBoundary THEN

PG.eState := E_PressureState.GaugeDisconnected; //Most likely not connected
PG.rPRESS := -1;

ELSE
	
PG.eState := OoR; //Larger voltage, probably out of range?
PG.rPRESS := -1;

END_IF


(* Pressure OK check *)
PG.xPRESS_OK := (PG.rPRESS >= MinPressure) AND (PG.eState >= 0);//Make sure to evaluate eState Too!!!!

(* Setpoint evaluation *)
PG.xAT_VAC := PG.xPRESS_OK AND (PG.rPRESS<PG.rVAC_SP);

END_FUNCTION_BLOCK

// ---- POUs/Functions/Gauge FB/FB_937A_VG.TcPOU
FUNCTION_BLOCK FB_937A_VG
VAR_IN_OUT
	VG : ST_VG;
END_VAR
VAR_INPUT
	PG	:	ST_VG := g_DummyVG;
END_VAR
VAR_OUTPUT
END_VAR
VAR
	rV	:	LREAL;
END_VAR

(* 937A Logarithmic Output Conversion *)
(* 7-15-2015 *)
(* This function will read the pressure from any gauge on a 937A. *)

rV := LREAL#10*INT_TO_LREAL(VG.iPRESS_R)/LREAL#32767;
VG.rPRESS := LREAL_TO_REAL(EXPT(10,rV/LREAL#0.6-LREAL#12));


(* Ion Gauge Protection Functions *)
(* If the PG pressure is greater than the VG.PRO_SP then the gauge is disabled *)
(* If the PG pressure is less than the VG.PRO_SP then the gauge is enabled *)
(* This FB also implements some hysteresis so the gauge doesn't have rapid power cycling while near the turn on boundary *)

IF PG.rPRESS < VG.rPRO_SP THEN

VG.xHV_DIS := NOT VG.xHV_SW;

ELSIF NOT VG.xHV_DIS THEN
	IF VG.rPRESS > VG.rPRO_SP + VG.rHYS_PR OR PG.rPRESS > VG.rPRO_SP + VG.rHYS_PR THEN
		VG.xHV_DIS := TRUE;
	END_IF
ELSE
	VG.xHV_DIS := TRUE;
END_IF


(* Pressure gauge OK checks *)
VG.xPRESS_OK := (rV <=9.6 ) AND (rV>=0.6); //legacy

IF (rV <=9.6 ) AND (rV>=0.6) THEN
	VG.eState := E_PressureState.Valid; // normal
ELSIF rV >= 0.18 AND rV <= 0.22 THEN
	VG.eState := E_PressureState.ValidLo; //LO
ELSIF rV >= 9.7 AND rV<= 9.9 THEN
	VG.eState := E_PressureState.ValidHi; //HIGH
ELSIF rV < 0.18 THEN
	VG.eState := E_PressureState.GaugeDisconnected; //not on
ELSE
	VG.eState := E_PressureState.PressInvalid; //other fault - could be no gauge, controller powering up etc
END_IF

(* Setpoint evaluation *)
VG.xAT_VAC := (VG.eState = E_PressureState.Valid) AND VG.rPRESS < VG.rVAC_SP;

END_FUNCTION_BLOCK

// ---- POUs/Functions/Gauge FB/FB_937B_VG.TcPOU
FUNCTION_BLOCK FB_937B_VG
VAR_IN_OUT
	VG : ST_VG;
END_VAR
VAR_INPUT
	PG	:	ST_VG := g_DummyVG;
END_VAR
VAR_OUTPUT
END_VAR
VAR
	rV	:	REAL;
END_VAR

(* 937B Logarithmic Output Conversion *)
(* 5-20-2016, Alex Wallace and Scott Stubbs *)
(* This function will read the pressure from any gauge on a 937B. *)

rV := 10*INT_TO_REAL(VG.iPRESS_R)/32767;
VG.rPRESS := LREAL_TO_REAL(EXPT(10,(rV-7.2)/0.6));


(* Ion Gauge Protection Functions *)
(* If the PG pressure is greater than the VG.PRO_SP then the gauge is disabled *)
(* If the PG pressure is less than the VG.PRO_SP then the gauge is enabled *)
(* This FB also implements some hysteresis so the gauge doesn't have rapid power cycling while near the turn on boundary *)

IF PG.rPRESS < VG.rPRO_SP THEN

VG.xHV_DIS := NOT VG.xHV_SW;

ELSIF NOT VG.xHV_DIS THEN
	IF VG.rPRESS > VG.rPRO_SP + VG.rHYS_PR OR PG.rPRESS > VG.rPRO_SP + VG.rHYS_PR THEN
		VG.xHV_DIS := TRUE;
	END_IF
ELSE
	VG.xHV_DIS := TRUE;
END_IF


(* Pressure gauge OK checks *)
VG.xPRESS_OK := (rV <=9.6 ) AND (rV>=0.6);

IF (rV <=9.7 ) AND (rV>=0.3) THEN
	VG.eState := Valid; // normal
ELSIF rV >= 0.18 AND rV <= 0.22 THEN
	VG.eState := ValidLo; //LO
ELSIF rV > 9.7 AND rV<= 9.9 THEN
	VG.eState := ValidHi; //HIGH
ELSIF rV < 0.18 THEN
	VG.eState := E_PressureState.GaugeDisconnected; //not on
ELSE
	VG.eState := PressInvalid; //other fault - could be no gauge, controller powering up etc
END_IF

(* Setpoint evaluation *)
VG.xAT_VAC := (VG.eState =Valid) AND VG.rPRESS < VG.rVAC_SP;

END_FUNCTION_BLOCK

// ---- POUs/Functions/Gauge FB/FB_972.TcPOU
FUNCTION_BLOCK FB_972
VAR_INPUT
END_VAR
VAR_OUTPUT
END_VAR
VAR_IN_OUT
	VG	: ST_VG;
END_VAR
VAR
	rV : LREAL;
END_VAR

(* Standard MKS 9XX series conversion *)
(* works for 972 and 925 *)

rV := 10*INT_TO_LREAL(VG.iPRESS_R)/32767;

IF rV > 1 THEN
	VG.rPRESS := LREAL_TO_REAL(EXPT(10, 2*rV-11));
	VG.xPRESS_OK := TRUE;
	VG.eState := Valid; //Press OK
ELSE
	VG.xPRESS_OK := FALSE;
	VG.eState := -6;
END_IF

END_FUNCTION_BLOCK

// ---- POUs/Functions/Gauge FB/FB_Dumb_Gauge.TcPOU
FUNCTION_BLOCK FB_Dumb_Gauge
VAR_IN_OUT
	iq_stPG : ST_VG;
END_VAR
VAR_INPUT
	i_stPGA : ST_VG;
	i_stPGB : ST_VG;
	i_stVRCA : ST_VRC;
	i_stVRCB : ST_VRC;
END_VAR
VAR_OUTPUT
END_VAR
VAR
END_VAR

(*
Alex Wallace 2013-10-28

The dummy gauge functions like so:
If my A side valve is open, I mimic the A side gauge.
If my B 	"	 			"			B	"		.
Else, I am at atmosphere, and my pressure is OK. 

The point of this gauge is to provide pressure readbacks for sections of the line that do not have gauges, and may move into an unknown pressure state.
*)

IF i_stVRCA.xOPN_DO THEN
iq_stPG := i_stPGA;
ELSIF i_stVRCB.xOPN_DO THEN
iq_stPG := i_stPGB;
ELSE
iq_stPG.xAT_VAC := FALSE;
iq_stPG.rPRESS := 750;
iq_stPG.xPRESS_OK := TRUE;
END_IF

END_FUNCTION_BLOCK

// ---- POUs/Functions/Pumps/FB_EbaraDryPump.TcPOU
FUNCTION_BLOCK FB_EbaraDryPump
VAR_INPUT
	i_stBPGauge	:	ST_VG; //booster pump interlock gauge
	i_xVlvOpn	:	BOOL; //valve(s) to main system load are open
END_VAR
VAR_OUTPUT
END_VAR
VAR_IN_OUT
	stPump	:	ST_EbaraDryPump; //Ebara dry pump structure
END_VAR
VAR
END_VAR

(* Ebara Dry Pump Control Routine
A. Wallace
2016-4-29
Applicable to:
EV-S20
EV-S50
EV-S100
EV-S200

Does basic controls for the pump. Starts booster pump when appropriate. Turns off pump
in the event of errors/ warnings. Provides interlocking interface.

Main Pump Operational Note:
Ebara recommends that the pump be exposed to the full system load after the main pump is running.

Booster Pump Operational Note:
The booster pump can either be started automatically by the pump itself (probably based on a timer?)
or it can be started by the PLC. The pressure setpoint is by default 30T. It may be wise to make
sure the pump was exposed to the full system load before starting the booster.

*)

//Mapping

// These are normally closed inputs
stPump.xErr := NOT stPump.i_xAlarm;
stPump.xWrn := NOT stPump.i_xWarning;


//Interlock and error/warning
stPump.xIlk :=  stPump.xExtIlk AND NOT (stPump.xErr OR stPump.xWrn);

//Start/ Stop the pump
IF stPump.xIlk THEN
	stPump.q_xMPStart := stPump.i_xRunSW;
ELSE
	stPump.q_xMPStart := stPump.i_xRunSW := FALSE;
END_IF

//Booster pump
stPump.xBPIlk := i_xVlvOpn AND stPump.i_xMPStatus AND (i_stBPGauge.rPRESS < stPump.rBPIlkSP) AND i_stBPGauge.xPRESS_OK;
stPump.tonBP(IN:=stPump.xBPIlk);
stPump.q_xBPStart := stPump.tonBP.Q;

END_FUNCTION_BLOCK

// ---- POUs/Functions/Pumps/FB_PTM_Pfeiffer.TcPOU
FUNCTION_BLOCK FB_PTM_Pfeiffer
VAR_IN_OUT
	iq_stPTM : ST_PfeifferPTM;
END_VAR
VAR_INPUT
END_VAR
VAR_OUTPUT
END_VAR
VAR
END_VAR

(* Basic pump supervisory section *)
IF iq_stPTM.xExtRunOk AND NOT (iq_stPTM.xFault OR iq_stPTM.i_xTempFault) THEN
	iq_stPTM.q_RunDO:=iq_stPTM.i_xRunSW;
ELSE
	iq_stPTM.i_xRunSW:=0;
	iq_stPTM.q_RunDO:=FALSE;
END_IF

END_FUNCTION_BLOCK

// ---- POUs/Functions/Pumps/FB_PTM_Ebara.TcPOU
FUNCTION_BLOCK FB_PTM_Ebara
VAR_IN_OUT
	iq_stPTM : ST_EbaraPTM;
END_VAR
VAR_INPUT
	i_iADCBits : UINT := 15;
	i_iRawSpeed: INT; //Should come from PLC Soft IO.
END_VAR
VAR_OUTPUT
END_VAR
VAR
	TOF_START: TOF := (PT:=T#0.5S); //Manual states momentary switches need to be closed for >= 0.3s
	TOF_STOP: TOF := (PT:=T#0.5S);
	TOF_RESET: TOF :=(PT:=T#0.5S);
END_VAR

(* Ebara ETC control FB
Scott Stubbs & Alex W.
*)

(* Switch processing *)
TOF_START.IN := iq_stPTM.i_xStart;
TOF_START();
TOF_STOP.IN  := iq_stPTM.i_xStop;
TOF_STOP();
TOF_RESET.IN := iq_stPTM.i_xReset;
TOF_RESET();

//Normally closed fault handling
iq_stPTM.xFault := NOT iq_stPTM.i_xNCFault;

(* Simple protection reset *)
IF iq_stPTM.xExtRunOk THEN
	iq_stPTM.q_xProtection:=TRUE;
END_IF

(* Basic pump supervisory section *)
	(* If override mode, ignore everything else *)
IF iq_stPTM.i_xOverride THEN
	IF TOF_START.Q THEN
	iq_stPTM.q_RunDO:=TRUE;
	ELSIF TOF_STOP.Q THEN
		iq_stPTM.q_RunDO:=FALSE;
	END_IF
	//Handle faults - the way the Ebara cable is done, xFault is normally closed
ELSIF iq_stPTM.xFault OR (iq_stPTM.q_RunDO AND NOT iq_stPTM.xExtRunOk) THEN
	iq_stPTM.q_RunDO:=FALSE;
	iq_stPTM.q_xProtection:=FALSE;
	//And one for when we need to start the pump normally. Only allows pump to be started if ILK ok.
ELSIF TOF_START.Q AND iq_stPTM.xExtRunOk THEN
	iq_stPTM.q_RunDO:=TRUE;
	iq_stPTM.q_xStart:=TOF_START.Q;
//One section for when pump is told to stop
ELSIF TOF_STOP.Q THEN
		iq_stPTM.q_RunDO:=FALSE;
END_IF 

iq_stPTM.q_xReset:=TOF_RESET.Q; //No need for a conditional on these, code below takes care of it
iq_stPTM.q_xStop:=TOF_STOP.Q;
//Reset the start switch after processing
IF iq_stPTM.q_RunDO THEN
	iq_stPTM.q_xStart := TOF_START.Q;
END_IF

(* Pump speed calculation *)
IF iq_stPTM.i_iRawSpeed / (EXPT(2,i_iADCBits)-1) * 10 >= 0.2 THEN //Speed reading appears to zero at ~0.16V
iq_stPTM.i_diCurSpd := LREAL_TO_DINT(iq_stPTM.i_iRawSpeed/(EXPT(2,i_iADCBits)-1)*67000);
//V (AI/(2^{# ADC bits} -1 ) * 10[ADC 10V scaling]) * (33600 [Max RPM] - 100) / 5
ELSE
	iq_stPTM.i_diCurSpd := 0;
END_IF

END_FUNCTION_BLOCK

// ---- POUs/Functions/Pumps/FB_PTM_Agilent.TcPOU
FUNCTION_BLOCK FB_PTM_Agilent
VAR_IN_OUT
	iq_stPTM	:	ST_AgilentPTM;
END_VAR
VAR_INPUT
END_VAR
VAR_OUTPUT
END_VAR
VAR
	
END_VAR

(* Basic Agilent Turbo Controls *)
(* A. Wallace, 2015-7-15 *)

(* Pump state *)
(* If frequency (R1) is not above setpoint and pump is not Starting, pump estate is STOPPED, 
   else if frequency (R1) is not above setpoint and pump is Starting, pump estate is STARTING, 
	else if frequency (R1) is above setpoint and pump is not Starting, pump estate is STOPPED, 
*)
IF iq_stPTM.xFault THEN 
	iq_stPTM.eState := E_PumpState.pumpFAULT;

ELSIF NOT iq_stPTM.i_xR1 AND NOT iq_stPTM.i_xSTART  THEN
	iq_stPTM.eState := E_PumpState.pumpSTOPPED;
ELSIF NOT iq_stPTM.i_xR1 AND iq_stPTM.i_xSTART  THEN
	iq_stPTM.eState := E_PumpState.pumpSTARTING;
ELSIF iq_stPTM.i_xR1 AND NOT iq_stPTM.i_xSTART THEN
	iq_stPTM.eState := E_PumpState.pumpRUNNING;
ELSE 
	iq_stPTM.eState := E_PumpState.pumpFAULT;
END_IF

(* Interlock Sum *)
iq_stPTM.q_xIlk := iq_stPTM.xExtRunOk AND NOT iq_stPTM.xFault;

(* Basic pump supervisory section *)
IF iq_stPTM.q_xIlk THEN
	iq_stPTM.q_RunDO := iq_stPTM.i_xRunSW;
ELSE
	iq_stPTM.i_xRunSW:=FALSE;
	iq_stPTM.q_RunDO:=FALSE;
END_IF

(* Mask the at speed bit if fault is true 
done for versions of the interface cable where
at speed gets its power from from the beckhoff term*)

(*Basically if Fault, then squash everything and turn everything off*)
IF iq_stPTM.xFault THEN
	iq_stPTM.i_xAtSpd := FALSE;
	iq_stPTM.i_xRunSW:=FALSE;
	iq_stPTM.q_RunDO:=FALSE;
	iq_stPTM.q_xSS := FALSE;
	iq_stPTM.q_xLSpd:= FALSE;
	iq_stPTM.eState := E_PumpState.pumpFAULT;
END_IF

END_FUNCTION_BLOCK

// ---- POUs/Functions/Pumps/FB_PTM_MagDriveDigital.TcPOU
FUNCTION_BLOCK FB_PTM_MagDriveDigital
VAR_IN_OUT
	iq_stPTM	:	ST_LeyboldPTM;
END_VAR
VAR_INPUT
END_VAR
VAR_OUTPUT
END_VAR
VAR
	xRunOk	:	BOOL;
	tofRemoteDelay	:	TOF;
	
END_VAR

(* Basic MagDrive Digital Turbo Controls *)
(* A. Wallace, 2015-7-15 *)

tofRemoteDelay(IN:=iq_stPTM.q_RunDO, PT:=T#5S);

iq_stPTM.q_xRemote := tofRemoteDelay.Q;

(* Interlock Sum *)
xRunOk := iq_stPTM.xExtRunOk AND NOT iq_stPTM.xFault;

(* Basic pump supervisory section *)
IF xRunOk THEN
	iq_stPTM.q_RunDO := iq_stPTM.i_xRunSW;
ELSE
	iq_stPTM.i_xRunSW:=FALSE;
	iq_stPTM.q_RunDO:=FALSE;
END_IF

END_FUNCTION_BLOCK

// ---- POUs/Functions/Pumps/FB_PTM_LeyboldTD20Classic.TcPOU
FUNCTION_BLOCK FB_PTM_LeyboldTD20Classic
VAR_IN_OUT
	iq_stPTM : ST_LeyboldPTM;
END_VAR
VAR_INPUT
END_VAR
VAR_OUTPUT
END_VAR
VAR
	rtReset	:	R_TRIG;
END_VAR

(* Leybold TD20 Classic FB
A. Wallace
NOTE: This FB should be instanced for each pump. It relies on a
persistent state for reseting faults.
*)

//Faults
	rtReset(CLK:=iq_stPTM.i_xReset);
	iq_stPTM.xFault R= rtReset.Q;
	iq_stPTM.xFault S= iq_stPTM.i_xTempFault OR NOT iq_stPTM.i_xNCError;

	iq_stPTM.xWarn R= rtReset.Q;
	iq_stPTM.xWarn S= iq_stPTM.xCommTimeout;

(* Basic pump supervisory section *)
IF iq_stPTM.xExtRunOk AND NOT iq_stPTM.xFault THEN
	iq_stPTM.q_RunDO:=iq_stPTM.i_xRunSW;
ELSE
	iq_stPTM.i_xRunSW:=FALSE;
	iq_stPTM.q_RunDO:=FALSE;
END_IF

END_FUNCTION_BLOCK

// ---- POUs/Functions/Pumps/FB_ScrollPump.TcPOU
FUNCTION_BLOCK FB_ScrollPump
VAR_IN_OUT
	iq_stPFO	:	ST_RoughPump;
END_VAR
VAR_INPUT
	TurboIsON : BOOL;
	VentValve	: ST_VCC_NO;
END_VAR
VAR
	Tmr_TOF : TOF;
END_VAR

//Turn on scroll pump if the Turbo Vent Valve is closed. So you are not just
// pumping air and accomplishing nothing

// cannot turn off scroll pump if turb is running. delay scroll off 150s.  


Tmr_TOF(IN:=TurboIsON, PT := T#150S);

IF VentValve.xCLS_DO THEN
	iq_stPFO.q_xRunDo := (Tmr_TOF.Q OR iq_stPFO.i_xRunSW);
ELSE
	iq_stPFO.q_xRunDo := FALSE;
END_IF

iq_stPFO.i_xRunSW := iq_stPFO.q_xRunDo;

END_FUNCTION_BLOCK

// ---- POUs/Functions/Pumps/FB_TurboExtLogic.TcPOU
FUNCTION_BLOCK FB_TurboExtLogic
VAR_IN_OUT
	Turbo		:	ST_AgilentPTM;
END_VAR
VAR_INPUT
	BackingGauge:	ST_VG;
	InletGauge	:	ST_VG;
	VentValve	:	ST_VCC_NO;
	ScrollPump	:	ST_RoughPump;
END_VAR
VAR_OUTPUT
END_VAR
VAR
END_VAR

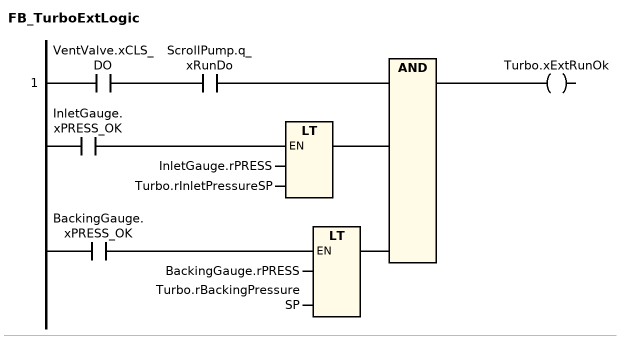
// NETWORK 1
Turbo.xExtRunOk := (VentValve.xCLS_DO AND ScrollPump.q_xRunDo) AND (InletGauge.xPRESS_OK AND InletGauge.rPRESS < Turbo.rInletPressureSP) AND (BackingGauge.xPRESS_OK AND BackingGauge.rPRESS < Turbo.rBackingPressureSP);

END_FUNCTION_BLOCK

// ---- POUs/Functions/Pumps/FB_VARIAN301TURBO.TcPOU
FUNCTION_BLOCK FB_VARIAN301TURBO

VAR_INPUT

	i_xglbAlmRst : BOOL;

END_VAR

VAR

	StartAlmTmr 	: TON;
	LSpdAlmTmr  	: TON;
	SSAlmTmr		: TON;
	tAlmDly			: TIME;

	xStartAlmFlag 	: BOOL;
	xLSpdAlmFlag  	: BOOL;
	xSSAlmFlag		: BOOL;

	xEND: BOOL;
END_VAR

VAR_IN_OUT

	iq_stTP: ST_PTM;

END_VAR

(* Resolve Interlocks *)
(* If Start Ilk is satisfied, other Ilk's are satisfied as well. *)

	iq_stTP.ilkEnb 	:= iq_stTP.ilkStart;
	iq_stTP.ilkLSpd	:= iq_stTP.ilkStart;
	iq_stTP.ilkSS	:= iq_stTP.ilkStart;

(* Hardware Enable Logic & Switch Feedback  *)
	IF NOT iq_stTP.ilkStart THEN
		iq_stTP.swStart := FALSE;
		iq_stTP.swLSpd := FALSE;
		iq_stTP.swSS := FALSE;
		iq_stTP.doEnb := FALSE;
	ELSE
		iq_stTP.doEnb := TRUE;
	END_IF;

(* Pump Control *)
	IF iq_stTP.doEnb THEN
		iq_stTP.doStart := iq_stTP.swStart;
		iq_stTP.doLSpd := iq_stTP.swLSpd;
		iq_stTP.doSS := iq_stTP.swSS;
	ELSE
		iq_stTP.doStart := FALSE;
		iq_stTP.doLSpd := FALSE;
		iq_stTP.doSS := FALSE;
	END_IF

(* ALARM SECTION *)
(* Standard Delay 30 minutes *)
tAlmDly := T#4m;

(* Fail To Start Alarm *)
xStartAlmFlag := iq_stTP.doStart AND NOT iq_stTP.diR1;
IF iq_stTP.doStart AND NOT iq_stTP.almStart THEN
	StartAlmTmr(IN:=xStartAlmFlag, PT:=tAlmDly, Q=>iq_stTP.almStart);
END_IF;
iq_stTP.AlmStart := iq_stTP.almStart AND NOT (i_xglbAlmRst OR iq_stTP.AlmRst);

(* Low Speed Failure Alarm *)
xLSpdAlmFlag := iq_stTP.doLSpd AND NOT iq_stTP.diLSpd;
IF iq_stTP.doLSpd AND NOT iq_stTP.almLSpd THEN
	LSpdAlmTmr(IN:=xLSpdAlmFlag, PT:=tAlmDly, Q=>iq_stTP.almLSpd);
END_IF;
iq_stTP.AlmLSpd := iq_stTP.AlmLSpd AND NOT (i_xglbAlmRst OR iq_stTP.AlmRst);

(* Soft Start Failure Alarm *)
xSSAlmFlag := iq_stTP.doSS AND NOT iq_stTP.diR1;
IF iq_stTP.doSS AND NOT iq_stTP.almSS THEN
	SSAlmTmr(IN:=xSSAlmFlag, PT:=tAlmDly, Q=>iq_stTP.almSS);
END_IF;
iq_stTP.AlmSS := iq_stTP.AlmSS AND NOT (i_xglbAlmRst OR iq_stTP.AlmRst);

(* Alarm Summary - Set the Alarm Summary flag if any alarm is active. *)
iq_stTP.AlmSum := iq_stTP.almFlt OR iq_stTP.almLSpd OR iq_stTP.AlmRst OR iq_stTP.almSS OR iq_stTP.almStart;

END_FUNCTION_BLOCK

// ---- POUs/Functions/Valve FB/FB_TurbVentvalve_NO.TcPOU
FUNCTION_BLOCK FB_TurbVentvalve_NO
VAR_IN_OUT
	iq_stValve : ST_VCC_NO;
END_VAR
VAR_INPUT
	i_stPTM	: ST_AgilentPTM;
END_VAR
VAR
	tofTmr 		: 	TOF;
END_VAR

(*If the turbo is on, you cannot open the valve. In order to open the valve, you have to allow the turbopump
 to have already been turned off for 2 minutes and you have to press the open button on the vent valve

If the code looks confusing please use a truth table to verify*)

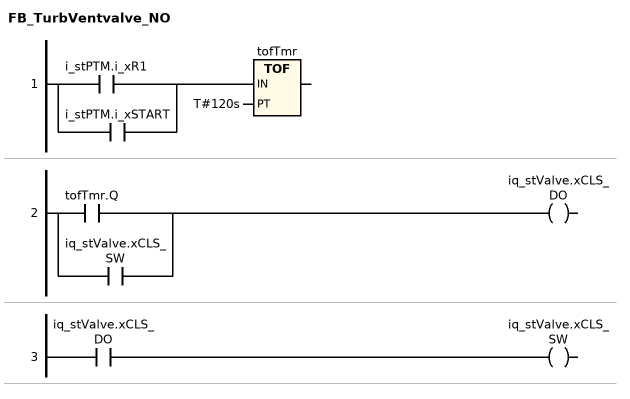
// NETWORK 1
tofTmr(IN := i_stPTM.i_xR1 OR i_stPTM.i_xSTART, PT := T#120s); // TOF

// NETWORK 2
iq_stValve.xCLS_DO := tofTmr.Q OR iq_stValve.xCLS_SW;

// NETWORK 3
iq_stValve.xCLS_SW := iq_stValve.xCLS_DO;

END_FUNCTION_BLOCK

// ---- POUs/Functions/Valve FB/FB_VCC_NO.TcPOU
FUNCTION_BLOCK FB_VCC_NO
VAR_IN_OUT

	iq_stValve : ST_VCC_NO;

END_VAR
VAR_INPUT

END_VAR
VAR_OUTPUT
END_VAR
VAR

tonOvrd	:	TON;
tonDelOK : TON;
rtOK	:	R_TRIG;

END_VAR


IF NOT iq_stValve.xCLS_OK THEN
iq_stValve.xCLS_SW := FALSE;
END_IF

(* Override logic *)
(* Goal: give ability to override, but do so in a way that people won't forget it.
Solution: Override only after ten seconds of override, protect against blips,
when the valve permission goes true for more than ten seconds consistently, remove override
*)

tonDelOK(IN:=iq_stValve.xCLS_OK, PT:=T#10S);
rtOK(CLK:=tonDelOK.Q);
IF rtOK.Q THEN iq_stValve.xOvrdCls :=FALSE; END_IF

//Override timer
tonOvrd(IN:=iq_stValve.xOvrdCls, PT:=T#10S);

(* Here's where the valve is closed *)
iq_stValve.xCLS_DO := (iq_stValve.xCLS_SW AND iq_stValve.xCLS_OK) OR (tonOvrd.Q AND g_stSystem.xOverrideMode);

END_FUNCTION_BLOCK

// ---- POUs/Functions/Valve FB/FB_VCN.TcPOU
FUNCTION_BLOCK FB_VCN
VAR_INPUT
	i_xExtIlk	:	BOOL; //External Interlock
	i_ReqPos	:	BOOL; //Requested position
END_VAR
VAR_OUTPUT
END_VAR
VAR_IN_OUT
	iq_stVCN	:	ST_VCN; //Needle valve structure
END_VAR
VAR
	// Requested voltage
	rReqVoltage: REAL := 0;
END_VAR
VAR CONSTANT
	rOpenVoltage	:	REAL := 9.1; // From the EVR 116 manual
	rCloseVoltage	:	REAL := 0.4;
END_VAR

(* Needle valve control FB
A. Wallace 2016-7-21

This FB should be used as a low level control block.

It provides:

Valve position ceiling
Interlock
Scaling

It is not intended for:
Closed-loop control

It could be used for:
Valve position/flow linearization

Note: Raw position calc is based on 0.5 to 9V span, 32767 bits
*)




// Interlocking
iq_stVCN.xIlk := i_xExtIlk;

IF iq_stVCN.xIlk THEN
	
	IF iq_stVCN.eValveControl = OpenValve THEN
		iq_stVCN.rReqPosition := iq_stVCN.rUpperLimit;
	ELSIF iq_stVCN.eValveControl = E_VCN.CloseValve THEN
		iq_stVCN.rReqPosition := 0;
	END_IF

	//Raw position calc
	iq_stVCN.rReqPosition := LIMIT(0, iq_stVCN.rReqPosition, iq_stVCN.rUpperLimit);
	rReqVoltage := iq_stVCN.rReqPosition * (rOpenVoltage-rCloseVoltage)/100 + rCloseVoltage;
	rReqVoltage := LIMIT(rCloseVoltage, rReqVoltage, rOpenVoltage); //The requested voltage should remain within this range
	iq_stVCN.q_iRawPosition := REAL_TO_INT( 32767/10 * rReqVoltage);	
ELSE
	iq_stVCN.q_iRawPosition := 0;
	iq_stVCN.rReqPosition := 0;
	iq_stVCN.eValveControl := E_VCN.CloseValve;
END_IF

END_FUNCTION_BLOCK

// ---- POUs/Functions/Valve FB/FB_VGC.TcPOU
FUNCTION_BLOCK FB_VGC
VAR_IN_OUT

	iq_stValve : ST_VGC;

END_VAR
VAR_INPUT

	i_stUSG	:	ST_VG;
	i_stDSG	:	ST_VG;

	i_xDis_DPIlk : BOOL := FALSE;  (* Set to true when calling the function to disable the differential pressure interlock *)
	rDiffPressAllowed	:	REAL := 22.5; // Torr, Default value comes from Vat Valve Manual
END_VAR
VAR_OUTPUT
END_VAR
VAR

	rDiffPress : REAL;
   set : BOOL;
   reset: Bool;
	  

	VGC_State : E_VGC;

	xFirstPass	:	BOOL;
	fbFSInit		:	R_TRIG;
	
	tonDelOK : TON;
	rtOK	:	R_TRIG;
	tonOvrd	:	TON;
	
	tDelOK	:	TIME := T#10S;
	tOvrd	:	TIME := T#10s;
END_VAR

(* Vacuum gate valve
A. Wallace
16-10-29

A gate valve isolates vacuum volumes. Ideally it can be opened when a system is vented
to allow for faster pumping, and will close when high vacuum is lost.

The following behavior is good for valves in something like a gas attenuator.
This function block does the following:
1. The valve can be opened when the difference between the pressures on both sides is
less than the maximum differential pressure.
2. This rule persists until the pressures on both sides are lower than the vacuum-setpoint.
3. Once at-vac, the valve will close if the pressure on either side rises above the setpoint.

Alternatively, the differential pressure interlock can be disabled so the valve may only be opened
if the pressure on both sides is lower than the at-vacuum-setpoint. You want this behavior if 
the valve is to be used in a UHV section.

Hysteresis is employed to ensure a smooth transition from vented/pumping down, to at-vac.

Finally, an override system is built in so you can bypass all the interlocking logic and 
get back online.
*)


fbFSInit( CLK := TRUE,
			Q => xFirstPass);

(* On first PLC pass, put valve into vented state, which implies a closed valve *)
IF xFirstPass THEN
VGC_State := E_VGC.Vented;
iq_stValve.xOPN_SW := FALSE;
END_IF

///Check valve postion
IF iq_stValve.i_xClsLS AND  iq_stValve.i_xOpnLS THEN
	iq_stValve.eState:=E_ValvePositionState.INVALID;
ELSIF NOT iq_stValve.i_xClsLS AND iq_stValve.i_xOpnLS THEN 
	iq_stValve.eState:=E_ValvePositionState.OPEN;
ELSIF iq_stValve.i_xClsLS AND NOT iq_stValve.i_xOpnLS THEN 
	iq_stValve.eState:=E_ValvePositionState.CLOSED;
ELSIF NOT iq_stValve.i_xClsLS AND NOT iq_stValve.i_xOpnLS THEN 
	iq_stValve.eState:=E_ValvePositionState.MOVING;
ELSE
	iq_stValve.eState:=E_ValvePositionState.INVALID;
END_IF

// Update hysteresis
IF iq_stValve.rAT_VAC_SP_LAST <> iq_stValve.rAT_VAC_SP OR xFirstPass THEN
	iq_stValve.rAT_VAC_SP_LAST := iq_stValve.rAT_VAC_SP;
	iq_stValve.rAT_VAC_HYS := iq_stValve.rHYST_PERC * iq_stValve.rAT_VAC_SP;
END_IF

iq_stValve.rAT_VAC_HYS := LIMIT(0, iq_stValve.rAT_VAC_HYS, iq_stValve.rAT_VAC_SP);
IF iq_stValve.rAT_VAC_SP <> 0 THEN
	IF iq_stValve.rHYST_PERC <> (iq_stValve.rAT_VAC_HYS / iq_stValve.rAT_VAC_SP) THEN
		iq_stValve.rHYST_PERC := LIMIT(0, (iq_stValve.rAT_VAC_HYS / iq_stValve.rAT_VAC_SP) ,1);
	END_IF
END_IF
// Valve at vacuum check
	set := i_stUSG.rPRESS < iq_stValve.rAT_VAC_HYS AND i_stDSG.rPRESS < iq_stValve.rAT_VAC_HYS AND i_stUSG.xPRESS_OK AND i_stDSG.xPRESS_OK;
 	iq_stValve.xAT_VAC S= set;
	reset := i_stUSG.rPRESS > iq_stValve.rAT_VAC_SP OR i_stDSG.rPRESS > iq_stValve.rAT_VAC_SP OR NOT i_stUSG.xPRESS_OK OR NOT i_stDSG.xPRESS_OK;
	iq_stValve.xAT_VAC R= reset;
	
// Differential pressure check
	(* Calc the differential pressure across the valve *)
	rDiffPress := ABS(i_stUSG.rPRESS - i_stDSG.rPRESS);
	
	(* As long as the differential pressure is less than 30mbar, the valve is allowed to open *)
	IF rDiffPress <= rDiffPressAllowed AND i_stUSG.xPRESS_OK AND i_stDSG.xPRESS_OK THEN
		iq_stValve.xDP_OK := TRUE;
	ELSE
		iq_stValve.xDP_OK	:= FALSE;
		(* If the differential pressure is exceeded, even when the valve is open,
		the state is unexpected and triggers a fault, because it suggests that something
		is wrong with the valve, or gauges or mapping or there is a major leak on one side.*)
		VGC_State := E_VGC.ERR_DiffPress;
	END_IF

// Valve state
CASE VGC_State OF
	E_VGC.Vented: (* The Vented state is used during pump down *)
		(* Assuming the pump down went well, we are now at vacuum on both sides,
		so we move to the vacuum state, otherwise remain in the vented state *)
		IF iq_stValve.xAT_VAC THEN
		VGC_State := E_VGC.AtVacuum;
		ELSE
		VGC_State := E_VGC.Vented;
		END_IF
	
	E_VGC.AtVacuum:
		IF iq_stValve.xAT_VAC THEN
		(* If both pressure setpoints are made,
		then enable the differential pressure interlock, regardless of the valve state
		assuming we're using some kind of ion gauge where a pressure setpoint cannot be higher than 1E-4 T *)
		VGC_State := E_VGC.AtVacuum;
		ELSE
		
			(* If the valve is open (or in an unknown state) and either gauge is not at it's vacuum setpoint,
			we have a loss of vacuum error *)
			IF (iq_stValve.i_xOpnLS OR (NOT iq_stValve.i_xOpnLS AND NOT iq_stValve.i_xClsLS)) THEN
			VGC_State := E_VGC.ERR_LostVac;
		
			(* Alternatively, if the valve is already closed and we lose pressure on one side,
			it was probably intentional venting, so we calmly move back to venting mode, and
			disable the differential pressure interlock *)
			ELSIF iq_stValve.i_xClsLS THEN
			VGC_State := E_VGC.Vented;
			END_IF
		
		END_IF
	
	E_VGC.ERR_DiffPress:
		VGC_State := E_VGC.Vented;
		iq_stValve.xERR_DifPres := TRUE;
	
	E_VGC.ERR_LostVac:
		VGC_State := E_VGC.Vented;
		iq_stValve.xERR_LstVac := TRUE;
	
ELSE
	VGC_State := E_VGC.Vented;
	iq_stValve.xERR_SM := TRUE;
	
END_CASE




// Interlock evaluation - with bypass for DP ILK bypass
IF i_xDis_DPIlk THEN
	iq_stValve.xOPN_OK := iq_stValve.xEXT_OK;
ELSE
	iq_stValve.xOPN_OK := iq_stValve.xEXT_OK AND iq_stValve.xAT_VAC;
END_IF


(* Valve operation *)

(* Reset the EPICS command to open the valve if the interlock is lost *)
IF NOT iq_stValve.xOPN_OK THEN
iq_stValve.xOPN_SW := FALSE;
END_IF

(* Override logic *)
(* Goal: give ability to override, but do so in a way that people won't forget it.
Solution: Override only after ten seconds of override, protect against blips,
when the valve permission goes true for more than ten seconds consistently, remove override
*)

tonDelOK(IN:=iq_stValve.xOPN_OK, PT:=tDelOK);
rtOK(CLK:=tonDelOK.Q);
IF rtOK.Q AND iq_stValve.xOvrdOpn THEN 
iq_stValve.xOvrdOpn :=FALSE;
iq_stValve.xOPN_SW := TRUE; //for seamless transition
END_IF

//Override timer
tonOvrd(IN:=iq_stValve.xOvrdOpn, PT:=tOvrd);

(* Here's where the valve opens *)
iq_stValve.xOPN_DO := (iq_stValve.xOPN_SW AND iq_stValve.xOPN_OK) OR (tonOvrd.Q AND g_stSystem.xOverrideMode);

// Alarm reset
ACT_ResetAlarms();

ACTION ACT_ResetAlarms:
iq_stValve.xERR_DifPres R= iq_stValve.xAlmRst;
iq_stValve.xERR_LstVac R= iq_stValve.xAlmRst;
END_ACTION

END_FUNCTION_BLOCK

// ---- POUs/Functions/Valve FB/FB_VGC_NO.TcPOU
FUNCTION_BLOCK FB_VGC_NO
VAR_IN_OUT

	iq_stValve : ST_VGC_NO;

END_VAR
VAR_INPUT

	i_stUSG	:	ST_VG;
	i_stDSG	:	ST_VG;

	i_xDis_DPIlk : BOOL := FALSE; (*Set to true when calling the function to disable the differential pressure interlock *)
	i_rDiffPressAllowed	:	REAL := 22.5;
END_VAR
VAR_OUTPUT
END_VAR
VAR

	rDiffPress : REAL;

	

	VGC_State : E_VGC;

	xFirstPass	:	BOOL;
	fbFSInit		:	R_TRIG;
	
	tonDelOK : TON;
	rtOK	:	R_TRIG;
	tonOvrd	:	TON;

END_VAR

(* Normally Open Gate Valve
This kind of gate valve can usually be found in systems with some kind of delicate window valve, not intended to hold
a full atmosphere.
*)

fbFSInit( CLK := TRUE,
			Q => xFirstPass);

(* On first PLC pass, put valve into vented state, which implies an open valve *)
IF xFirstPass THEN
VGC_State := E_VGC.Vented;
iq_stValve.xCLS_SW := FALSE;
END_IF

///Check valve postion
IF NOT iq_stValve.i_xClsLS AND iq_stValve.i_xOpnLS THEN 
	iq_stValve.eState:=E_ValvePositionState.OPEN;
ELSIF iq_stValve.i_xClsLS AND NOT iq_stValve.i_xOpnLS THEN 
	iq_stValve.eState:=E_ValvePositionState.CLOSED;
ELSIF NOT iq_stValve.i_xClsLS AND NOT iq_stValve.i_xOpnLS THEN 
	iq_stValve.eState:=E_ValvePositionState.MOVING;
ELSE
	iq_stValve.eState:=E_ValvePositionState.INVALID;
END_IF

(* Calc the differential pressure across the valve *)
rDiffPress := ABS(i_stUSG.rPRESS - i_stDSG.rPRESS);


(* Here's where the Dis_DPIlk can enable or disable the DP interlock code above,
By default the Dis_DPIlk is FALSE, so the valve is interlocked by the external interlocks
and the differential pressure across the valve. *)

IF i_xDis_DPIlk THEN
iq_stValve.xCLS_OK := iq_stValve.xEXT_OK;
ELSE

CASE VGC_State OF

E_VGC.Vented: (* The Vented state is used during pump down *)
	
	(* As long as the differential pressure is less than 30mbar, the valve is allowed to close/ remain closed *)
	IF rDiffPress <= i_rDiffPressAllowed AND i_stUSG.xPRESS_OK AND i_stDSG.xPRESS_OK THEN
	iq_stValve.xDP_OK := TRUE;
	ELSE
	iq_stValve.xDP_OK	:= FALSE;
	(* If the differential pressure is exceeded, even when the valve is open,
	the state is unexpected and triggers a fault, because it suggests that something
	is wrong with the valve, or gauges or mapping or there is a major leak on one side.*)
	VGC_State := E_VGC.ERR_DiffPress;
	END_IF
	
	(* Assuming the pump down went well, we are now at vacuum on both sides,
	so we move to the vacuum state, otherwise remain in the vented state *)
	IF i_stUSG.xAT_VAC AND i_stDSG.xAT_VAC AND i_stUSG.xPRESS_OK AND i_stDSG.xPRESS_OK THEN
	VGC_State := E_VGC.AtVacuum;
	ELSE
	VGC_State := E_VGC.Vented;
	END_IF

E_VGC.AtVacuum:
	(* Note for normally open valves, the condition for remaining closed is that the differential pressure
	does not exceed some certain value, which comes from the pressure that the window can hold.
	*)
	IF rDiffPress <= i_rDiffPressAllowed AND i_stUSG.xPRESS_OK AND i_stDSG.xPRESS_OK THEN
	(* If both pressure setpoints are made,
	then enable the differential pressure interlock, regardless of the valve state
	assuming we're using some kind of ion gauge where a pressure setpoint cannot be higher than 1E-4 T *)
	iq_stValve.xDP_OK := TRUE;
	VGC_State := E_VGC.AtVacuum;
	ELSE
	
		(* If the valve is closed (or in an unknown state) and either gauge is not at it's vacuum setpoint,
		we have a loss of vacuum error *)
		IF (iq_stValve.i_xClsLS OR (NOT iq_stValve.i_xOpnLS AND NOT iq_stValve.i_xClsLS)) AND 
		(NOT i_stUSG.xAT_VAC OR NOT i_stDSG.xAT_VAC) THEN
			VGC_State := E_VGC.ERR_LostVac;
			iq_stValve.xDP_OK := FALSE;
	
		(* Alternatively, if the valve is already open and we lose vacuum or differential pressure,
		it was probably intentional venting, so we calmly move back to venting mode, and
		disable the differential pressure interlock *)
		ELSIF iq_stValve.i_xOpnLS AND(NOT i_stUSG.xAT_VAC OR NOT i_stDSG.xAT_VAC) THEN
			iq_stValve.xDP_OK := FALSE;
			VGC_State := E_VGC.Vented;
		END_IF
	
	END_IF

E_VGC.ERR_DiffPress:
	iq_stValve.xDP_OK := FALSE;
	VGC_State := E_VGC.Vented;
	iq_stValve.xERR_DifPres := TRUE;

E_VGC.ERR_LostVac:
	iq_stValve.xDP_OK := FALSE;
	VGC_State := E_VGC.Vented;
	iq_stValve.xERR_LstVac := TRUE;
	
ELSE
	VGC_State := E_VGC.Vented;
	iq_stValve.xERR_SM := TRUE;

END_CASE

(* In the default state the Valve.CLS_OK depends on both the external and differential pressure interlocks *)
iq_stValve.xCLS_OK := iq_stValve.xEXT_OK AND iq_stValve.xDP_OK;
END_IF

(* Valve operation *)

(* Reset the PLC/EPICS command to open the valve if the interlock is lost *)
IF NOT iq_stValve.xCLS_OK THEN
iq_stValve.xCLS_SW := FALSE;
END_IF

(* Override logic *)
(* Goal: give ability to override, but do so in a way that people won't forget it.
Solution: Override only after ten seconds of override, protect against blips,
when the valve permission goes true for more than ten seconds consistently, remove override
*)

tonDelOK(IN:=iq_stValve.xCLS_OK, PT:=T#10S);
rtOK(CLK:=tonDelOK.Q);
IF rtOK.Q AND iq_stValve.xOvrdCls THEN 
iq_stValve.xOvrdCls :=FALSE;
iq_stValve.xCLS_SW := TRUE;
END_IF

//Override timer
tonOvrd(IN:=iq_stValve.xOvrdCls, PT:=T#10S);

(* Here's where the valve is closed *)
iq_stValve.xCLS_DO := (iq_stValve.xCLS_SW AND iq_stValve.xCLS_OK) OR (tonOvrd.Q AND g_stSystem.xOverrideMode);

ACTION ACT_ResetAlarms:
iq_stValve.xERR_DifPres R= iq_stValve.xAlmRst;
iq_stValve.xERR_LstVac R= iq_stValve.xAlmRst;
END_ACTION

END_FUNCTION_BLOCK

// ---- POUs/Functions/Valve FB/FB_VRC.TcPOU
FUNCTION_BLOCK FB_VRC
VAR_IN_OUT

	iq_stValve : ST_VRC;

END_VAR
VAR_INPUT

END_VAR
VAR_OUTPUT
END_VAR
VAR

tonOvrd	:	TON;
tonDelOK : TON;
rtOK	:	R_TRIG;

END_VAR


///Check valve postion
IF NOT iq_stValve.i_xClsLS AND iq_stValve.i_xOpnLS THEN 
	iq_stValve.eState:=E_ValvePositionState.OPEN;
ELSIF iq_stValve.i_xClsLS AND NOT iq_stValve.i_xOpnLS THEN 
	iq_stValve.eState:=E_ValvePositionState.CLOSED;
ELSIF NOT iq_stValve.i_xClsLS AND NOT iq_stValve.i_xOpnLS THEN 
	iq_stValve.eState:=E_ValvePositionState.MOVING;
ELSE
	iq_stValve.eState:=E_ValvePositionState.INVALID;
END_IF

IF NOT iq_stValve.xOPN_OK and NOT tonOvrd.Q THEN
iq_stValve.xOPN_SW := FALSE;
END_IF

(* Override logic *)
(* Goal: give ability to override, but do so in a way that people won't forget it.
Solution: Override only after ten seconds of override, protect against blips,
when the valve permission goes true for more than ten seconds consistently, remove override
*)

tonDelOK(IN:=iq_stValve.xOPN_OK, PT:=T#10S);
rtOK(CLK:=tonDelOK.Q);
IF rtOK.Q THEN iq_stValve.xOvrdOpn :=FALSE; END_IF

//Override timer
tonOvrd(IN:=iq_stValve.xOvrdOpn, PT:=T#10S);

(* Here's where the valve opens *)
iq_stValve.xOPN_DO := (iq_stValve.xOPN_SW AND iq_stValve.xOPN_OK) OR (tonOvrd.Q AND g_stSystem.xOverrideMode);

END_FUNCTION_BLOCK

// ---- POUs/Functions/Valve FB/FB_VCC.TcPOU
FUNCTION_BLOCK FB_VCC
VAR_IN_OUT

	iq_stValve : ST_VCC;

END_VAR
VAR_INPUT

END_VAR
VAR_OUTPUT
END_VAR
VAR

tonOvrd	:	TON;
tonDelOK : TON;
rtOK	:	R_TRIG;

END_VAR


IF NOT iq_stValve.xOPN_OK THEN
iq_stValve.xOPN_SW := FALSE;
END_IF

(* Override logic *)
(* Goal: give ability to override, but do so in a way that people won't forget it.
Solution: Override only after ten seconds of override, protect against blips,
when the valve permission goes true for more than ten seconds consistently, remove override
*)

tonDelOK(IN:=iq_stValve.xOPN_OK, PT:=T#10S);
rtOK(CLK:=tonDelOK.Q);
IF rtOK.Q THEN iq_stValve.xOvrdOpn :=FALSE; END_IF

//Override timer
tonOvrd(IN:=iq_stValve.xOvrdOpn, PT:=T#10S);

(* Here's where the valve opens *)
iq_stValve.xOPN_DO := (iq_stValve.xOPN_SW AND iq_stValve.xOPN_OK) OR (tonOvrd.Q AND g_stSystem.xOverrideMode);

END_FUNCTION_BLOCK

// ---- POUs/Functions/Valve FB/FB_VRC_OK_CLS.TcPOU
FUNCTION_BLOCK FB_VRC_OK_CLS
VAR_IN_OUT

	iq_stValve : ST_VRC;

END_VAR
VAR_INPUT

END_VAR
VAR_OUTPUT
END_VAR
VAR

tonOvrd	:	TON;
tonDelOK : TON;
rtOK	:	R_TRIG;

END_VAR

(* This fumction block is different from the regular VRC in that CLOSING must be permitted. *)
(* Implemented for the funky valve 04 on LAMP *)
IF NOT iq_stValve.xOPN_OK and NOT tonOvrd.Q THEN
iq_stValve.xOPN_SW := FALSE;
END_IF

(* Override logic *)
(* Goal: give ability to override, but do so in a way that people won't forget it.
Solution: Override only after ten seconds of override, protect against blips,
when the valve permission goes true for more than ten seconds consistently, remove override
*)

tonDelOK(IN:=iq_stValve.xOPN_OK, PT:=T#10S);
rtOK(CLK:=tonDelOK.Q);
IF rtOK.Q THEN iq_stValve.xOvrdOpn :=FALSE; END_IF

//Override timer
tonOvrd(IN:=iq_stValve.xOvrdOpn, PT:=T#10S);

(* Here's where the valve opens *)
iq_stValve.xOPN_DO := NOT iq_stValve.xCLS_OK OR ((iq_stValve.xOPN_SW AND iq_stValve.xOPN_OK) OR (tonOvrd.Q AND g_stSystem.xOverrideMode));

END_FUNCTION_BLOCK

// ---- POUs/Functions/Valve FB/F_VALVE_REL_ILK.TcPOU
FUNCTION F_VALVE_REL_ILK : BOOL
VAR_INPUT
	i_stUSG	:	ST_VG;
	i_stDSG	:	ST_VG;
	//Orders of magnitude allowed between up/downstream pressures for valve to open. Must be real positive integer.
	i_iOrdersMagnitude: INT;
END_VAR
VAR
	rPressRatio : REAL;
	rMaxRatioAllowed	:	LREAL := EXPT(10,INT_TO_LREAL(i_iOrdersMagnitude));
	rMinRatioAllowed	:	LREAL := EXPT(10,INT_TO_LREAL(-1 * i_iOrdersMagnitude));
END_VAR

(* S. Stubbs 11/2015 *)

(* OK, this is going to be a general-use function that will return whether the ratio of the pressures given is less than x orders of magnitude.
True iff 10^(-x) < a/b < 10^x.  Simple, right?  Just make sure it gets a positive order of magnitude and the pressures aren't 0. ~Scott *)   

(* Find ratio *)

IF i_stDSG.rPRESS <> 0 THEN
	rPressRatio := i_stUSG.rPRESS / i_stDSG.rPRESS;

	F_VALVE_REL_ILK := rPressRatio < rMaxRatioAllowed AND rMinRatioAllowed < rPressRatio;
ELSE
	F_VALVE_REL_ILK := FALSE;
END_IF

END_FUNCTION

// ---- POUs/Functions/Valve FB/F_VRC_DIODE_ILK.TcPOU
FUNCTION F_VRC_DIODE_ILK : BOOL
VAR_INPUT

	i_stPGA : ST_VG;
	i_stPGB	: ST_VG;

END_VAR
VAR

	rHysterisis : REAL := 0;

	xInterlock: BOOL;
	rTolerance: REAL := 20;
END_VAR

(* The principle is simple, a VRC should never open when B side pressure is greater than the A side pressure. *)
rTolerance := 20;
F_VRC_DIODE_ILK := ((i_stPGA.rPRESS + rTolerance >= i_stPGB.rPRESS + rHysterisis) OR i_stPGA.xBAKEOUT) AND i_stPGA.xPRESS_OK AND i_stPGB.xPRESS_OK;

(* OK it gets a bit more complicated with hysterisis,

Now, if the F_VIC_DIODE_ILK is FALSE then some hysterisis is added to the B side. But if it's OK then we just stick with making sure that the A side is greater than the B side

*)

END_FUNCTION

// ---- POUs/Functions/Valve FB/F_TURBO_VRC_ILK.TcPOU
FUNCTION F_TURBO_VRC_ILK : BOOL
VAR_INPUT

	i_xHiVac 	: BOOL;
	i_xRunPTM	: BOOL;
	i_xFLVac	: BOOL;

END_VAR
VAR

	rHysterisis : REAL := 0;

	xInterlock: BOOL;
	rTolerance: REAL := 20;
END_VAR

(* Close the vic if the roughing pump pirani loses its at-vac setpoint while the turbo is pumping *)
F_TURBO_VRC_ILK := (NOT i_xHiVac AND NOT i_xRunPTM AND NOT i_xFLVac) OR
					(NOT i_xRunPTM AND i_xFLVac) OR
					(i_xRunPTM AND i_xFLVac);

END_FUNCTION
